(* IEC 61131-3 sources: Yaha/Documentation/Infomaterial/OSCAT/pcworx_basic_333/module_export (part 5) *)

(* ---- MATRIX.ST ---- *)
(*@PROPERTIES_EX@
TYPE: POU
LOCALE: 0
IEC_LANGUAGE: ST
PLC_TYPE: independent
PROC_TYPE: independent
GROUP: LOGIC.OTHER
*)
(*@KEY@:DESCRIPTION*)
version 1.3	26 oct. 2008
programmer 	hugo
tested by	oscat

MATRIX is a matrix keyboard encoder for 4 rows and up to 5 columns.
matrix can send a code while a key is pressed and it sends another code while a key is released when the setup variable 'release' is set to true.
the setup variable release is false the code is only sent when the key is pressed.
the output byte holds the 5 columns in the lowest bits 0..2  and the row number in bits 4..6, while bit 7 is true for a key pressed and false for a key released.
(*@KEY@:END_DESCRIPTION*)
FUNCTION_BLOCK MATRIX

(*Group:Default*)

VAR_INPUT
	X1 :	BOOL;
	X2 :	BOOL;
	X3 :	BOOL;
	X4 :	BOOL;
	X5 :	BOOL;
	RELEASE :	BOOL;
END_VAR

VAR_OUTPUT
	CODE :	BYTE;
	TP :	BOOL;
	Y1 :	BOOL := TRUE;
	Y2 :	BOOL;
	Y3 :	BOOL;
	Y4 :	BOOL;
END_VAR

VAR
	line :	BYTE;
	X :	oscat_arb_0_3;(*scan line inputs*)
	L :	oscat_arb_0_3;(*scan line status*)
	i :	INT;
	temp :	BYTE;
	temp2 :	BYTE;
	L_temp :	BYTE;
	temp_bit :	BOOL;
	in_temp :	INT;
END_VAR

(*@KEY@: WORKSHEET
NAME: MATRIX
IEC_LANGUAGE: ST
*)
TP := FALSE;
code := BYTE#0;

(* read scan lines *)
in_temp := _BYTE_TO_INT(line);
temp := X[in_temp];  (* X[LINE] umkopieren *)

temp:=BIT_LOAD_B(temp,X1,0); (* X[line].0 := X1; *)
temp:=BIT_LOAD_B(temp,X2,1); (* X[line].1 := X2; *)
temp:=BIT_LOAD_B(temp,X3,2); (* X[line].2 := X3; *)
temp:=BIT_LOAD_B(temp,X4,3); (* X[line].3 := X4; *)
temp:=BIT_LOAD_B(temp,X5,4); (* X[line].4 := X5; *)

X[in_temp] := temp; (* X[LINE] zurückkopieren *)

(* compare for change *)
FOR i := 0 TO 3 DO
	IF X[i] <> L[i] THEN
		(* scan line information has changed code need to be found and generated *)
		temp   := x[i] XOR L[i];
        temp2  := X[i];
        L_temp := L[i];

        IF BIT_OF_DWORD(BYTE_TO_DWORD(temp),0) THEN (* temp.X0 *)
			code := BYTE#1;
            temp_bit := BIT_OF_DWORD(BYTE_TO_DWORD(temp2),0);   (* X[i].X0 *)
            code := BIT_LOAD_B(code,temp_bit,7);     			(* code.X7 *)
            L_temp := BIT_LOAD_B(L_temp,temp_bit,0); 			(* L[i].X0 *)
		ELSIF BIT_OF_DWORD(BYTE_TO_DWORD(temp),1) THEN          (* temp.X1 *)
			code := BYTE#2;
            temp_bit := BIT_OF_DWORD(BYTE_TO_DWORD(temp2),1);   (* X[i].X1 *)
            code := BIT_LOAD_B(code,temp_bit,7);     			(* code.X7 *)
            L_temp := BIT_LOAD_B(L_temp,temp_bit,1); 			(* L[i].X1 *)
		ELSIF BIT_OF_DWORD(BYTE_TO_DWORD(temp),2) THEN          (* temp.X2 *)
			code := BYTE#3;
            temp_bit := BIT_OF_DWORD(BYTE_TO_DWORD(temp2),2);   (* X[i].X2 *)
            code := BIT_LOAD_B(code,temp_bit,7);     			(* code.X7 *)
            L_temp := BIT_LOAD_B(L_temp,temp_bit,2); 			(* L[i].X2 *)
		ELSIF BIT_OF_DWORD(BYTE_TO_DWORD(temp),3) THEN          (* temp.X3 *)
			code := BYTE#4;
            temp_bit := BIT_OF_DWORD(BYTE_TO_DWORD(temp2),3);   (* X[i].X3 *)
            code := BIT_LOAD_B(code,temp_bit,7);     			(* code.X7 *)
            L_temp := BIT_LOAD_B(L_temp,temp_bit,3); 			(* L[i].X3 *)
		ELSIF BIT_OF_DWORD(BYTE_TO_DWORD(temp),4) THEN          (* temp.X4 *)
			code := BYTE#5;
            temp_bit := BIT_OF_DWORD(BYTE_TO_DWORD(temp2),4);   (* X[i].X4 *)
            code := BIT_LOAD_B(code,temp_bit,7);     			(* code.X7 *)
            L_temp := BIT_LOAD_B(L_temp,temp_bit,4); 			(* L[i].X4 *)
		END_IF;
        L[i] := L_temp;
		TP := TRUE;
        code := (code AND BYTE#2#1000_1111) OR SHL(LINE AND BYTE#2#0000_0111,4);
        (* obere zeile enspricht: Code.X4 := Line.X0; /  Code.X5 := Line.X1; / Code.X6 := Line.X2; *)

		(* check if release codes need to be killed *)
		IF NOT release AND code < BYTE#127 THEN
			code := BYTE#0;
			TP := FALSE;
		END_IF;
        EXIT;
	END_IF;
END_FOR;

(* increment scan line every cycle *)
line := INT_TO_BYTE(_BYTE_TO_INT(line) + 1) AND BYTE#2#0000_0011;
temp := SHL(BYTE#1,_BYTE_TO_INT(line));

Y1 := BIT_OF_DWORD(BYTE_TO_DWORD(temp),0); (* temp.0 *)
Y2 := BIT_OF_DWORD(BYTE_TO_DWORD(temp),1); (* temp.1 *)
Y3 := BIT_OF_DWORD(BYTE_TO_DWORD(temp),2); (* temp.2 *)
Y4 := BIT_OF_DWORD(BYTE_TO_DWORD(temp),3); (* temp.3 *)

(* revision history
hm		10.6.2007	rev 1.0
	original version

hm		11.9.2007	rev 1.1
	deleted unused variables k and old_code

hm		23.12.2007	rev 1.2
	added exit statement in for loop instead of i:=5

hm		26. oct. 2008	rev 1.3
	code optimized

*)
(*@KEY@: END_WORKSHEET *)
END_FUNCTION_BLOCK

(* ---- MESSAGE_4R.ST ---- *)
(*@PROPERTIES_EX@
TYPE: POU
LOCALE: 0
IEC_LANGUAGE: ST
PLC_TYPE: independent
PROC_TYPE: independent
GROUP: STRINGS
*)
(*@KEY@:DESCRIPTION*)
version 1.1	27. oct. 2008
programmer 	hugo
tested by	tobias

this function generates a rotation meassage with up to 4 strings.
on each rising edge of EN the next message in line will be displayed.
when EN stays high longer then one cycle, the next message will be displayed automatically after the time T1 is elapsed.
the output MX is the generated message and CX is a counter 0..3 signaling the current message displayed.
the displayed messages are 0 .. MM.
(*@KEY@:END_DESCRIPTION*)
FUNCTION_BLOCK MESSAGE_4R

(*Group:Default*)

VAR_INPUT
	M0 :	STRING;
	M1 :	STRING;
	M2 :	STRING;
	M3 :	STRING;
	MM :	INT := 3;
	ENQ :	BOOL := TRUE;
	CLK :	BOOL := TRUE;
	T1 :	TIME := T#3s;
END_VAR

VAR_OUTPUT
	MX :	STRING;
	MN :	INT;
	TR :	BOOL;
END_VAR

VAR
	timer :	TON;
	edge :	BOOL;
END_VAR

(*@KEY@: WORKSHEET
NAME: MESSAGE_4R
IEC_LANGUAGE: ST
*)
(* check for rising edge on EN *)
TR := FALSE;
IF ENQ THEN
	IF (NOT edge AND clk) OR timer.q THEN
			MN := INC1(MN, MM);
			TR := TRUE;
			timer(in := FALSE);
			CASE MN OF
				0 : MX := M0;
				1 : MX := M1;
				2 : MX := M2;
				3 : MX := M3;
			END_CASE;
	END_IF;
	edge := clk;
	timer( in := CLK, pt := T1);
ELSE
	MX := '';
	MN := 0;
END_IF;

(* revision history
hm	8. oct. 2008	rev 1.0
	original version

hm	27. oct. 2008	rev 1.1
	changed _INC to INC1

*)
(*@KEY@: END_WORKSHEET *)
END_FUNCTION_BLOCK

(* ---- MESSAGE_8.ST ---- *)
(*@PROPERTIES_EX@
TYPE: POU
LOCALE: 0
IEC_LANGUAGE: ST
PLC_TYPE: independent
PROC_TYPE: independent
GROUP: STRINGS
*)
(*@KEY@:DESCRIPTION*)
version 1.1	29. mar. 2008
programmer 	hugo
tested by	tobias

this function generates one out of 4 messages specified by S1 .. S8.
the selected message will be presented at the output M.
In1 has higher priority then In2 which has higher priority then IN3 and in8 has the lowest priority.
(*@KEY@:END_DESCRIPTION*)
FUNCTION_BLOCK MESSAGE_8

(*Group:Default*)

VAR_INPUT
	IN1 :	BOOL;
	IN2 :	BOOL;
	IN3 :	BOOL;
	IN4 :	BOOL;
	IN5 :	BOOL;
	IN6 :	BOOL;
	IN7 :	BOOL;
	IN8 :	BOOL;
	S1 :	STRING;
	S2 :	STRING;
	S3 :	STRING;
	S4 :	STRING;
	S5 :	STRING;
	S6 :	STRING;
	S7 :	STRING;
	S8 :	STRING;
END_VAR

VAR_OUTPUT
	M :	STRING;
END_VAR

(*@KEY@: WORKSHEET
NAME: MESSAGE_8
IEC_LANGUAGE: ST
*)
(* check if an alarm is present if yes set the output M otherwise clear M *)
IF in1 THEN
	M := S1;
ELSIF in2 THEN
	M := S2;
ELSIF in3 THEN
	M := S3;
ELSIF in4 THEN
	M := S4;
ELSIF in5 THEN
	M := S5;
ELSIF in6 THEN
	M := S6;
ELSIF in7 THEN
	M := S7;
ELSIF in8 THEN
	M := S8;
ELSE
	M := '';
END_IF;

(* revision history
hm	26.12.2007		rev 1.0
	original version

hm	29. mar. 2008	rev 1.1
	changed STRING to STRING(STRING_LENGTH)
*)
(*@KEY@: END_WORKSHEET *)
END_FUNCTION_BLOCK

(* ---- METER.ST ---- *)
(*@PROPERTIES_EX@
TYPE: POU
LOCALE: 0
IEC_LANGUAGE: ST
PLC_TYPE: independent
PROC_TYPE: independent
GROUP: ENGINEERING.MEASUREMENTS
*)
(*@KEY@:DESCRIPTION*)
version 1.4	8. mar. 2009
programmer 	oscat
tested BY	oscat

METER measures usage of power or similar values the output MX is the sum of the inputs over time.
MX := sum over time of (I1 * P1 + I2 * P2)/D.
a simple example is the consumption counter for a 2 stage oil burner where stage 1 is 10KW and stage 2 is 20KW.
I1 and I2 decide which value is accounted for, I1 = True only counts P1, I2 is True counts P2
and I1 and I2 is true counts P1 and P2.
the meter can be used for all kind of consumption meters. P1 and P2 can change on the fly.

(*@KEY@:END_DESCRIPTION*)
FUNCTION_BLOCK METER

(*Group:Default*)

VAR_INPUT
	M1 :	REAL;
	M2 :	REAL;
	I1 :	BOOL;
	I2 :	BOOL;
	D :	REAL := 1.0;
	RST :	BOOL;
END_VAR

VAR_IN_OUT
	MX :	REAL;
END_VAR

VAR RETAIN
	MR :	REAL2;
END_VAR

VAR
	MX1 :	REAL;(*current consumption value on M1 and M2*)
	MX2 :	REAL;(*current consumption value on M1 and M2*)
	tx :	UDINT;
	last :	UDINT;
	tc :	REAL;
	init :	BOOL;
	T_PLC_MS :	T_PLC_MS;
	R2_ADD :	R2_ADD;
END_VAR

(*@KEY@: WORKSHEET
NAME: METER
IEC_LANGUAGE: ST
*)
(* measure the last cycle time and make sure we onle execute once every millisecond *)
T_PLC_MS();
tx:= T_PLC_MS.T_PLC_MS;
IF NOT init THEN
	init := TRUE;
	last := tx;
	mr.RX := mx;
	mr.R1 := 0.0;
ELSIF tx = last THEN
	RETURN;
ELSE
	tc := UDINT_TO_REAL(tx - last) * 0.001;
END_IF;
last := tx;

(* reset *)
IF rst THEN
	mr.R1 := 0.0;
	mr.RX := 0.0;
ELSE
	(* current consumption measurement *)
	MX1 := SEL(I1,0.0,M1);
	MX2 := SEL(I2,0.0,M2);
	(* add up the current values in a double real *)
	R2_ADD(X:=MR,Y:=(SEL(I1,0.0,mx1) + SEL(I2, 0.0, mx2)) / D * TC);
	MR:=R2_ADD.R2_ADD;
	(* set the current output value *)
	MX := mr.RX;
END_IF;

(* revision history

hm	16. sep.2007		rev 1.0
	original version

hm	7. feb 2008		rev 1.1
	use new version of ft_int to avoid a counting stop at high values
	deleted unnecessary limits

hm	24. mar. 2008		rev 1.2
	use data_type real2 to extend accuracy to 15 digits total
	do not use ft_int which adds unnecessary overhead

hm	8. feb. 2009		rev 1.3
	changed mx to be I/O
	make sure calculation works for cycle times < 1 ms

hm	8. mar. 2009	rev 1.4
	last was not updated
	code improvements

*)

(*@KEY@: END_WORKSHEET *)
END_FUNCTION_BLOCK

(* ---- METER_STAT.ST ---- *)
(*@PROPERTIES_EX@
TYPE: POU
LOCALE: 0
IEC_LANGUAGE: ST
PLC_TYPE: independent
PROC_TYPE: independent
GROUP: ENGINEERING.MEASUREMENTS
*)
(*@KEY@:DESCRIPTION*)
version 1.3	18. jul. 2009
programmer 	oscat
tested BY	oscat

METER_STAT runs statistics of a metered value, it calculates the current week, day, month and year consumption and stores the corresponding last day, week, month and year value.

(*@KEY@:END_DESCRIPTION*)
FUNCTION_BLOCK METER_STAT

(*Group:Default*)

VAR_INPUT
	IN :	REAL;
	DI :	UDINT;
	RST :	BOOL;
END_VAR

VAR_IN_OUT
	LAST_DAY :	REAL;
	CURRENT_DAY :	REAL;
	LAST_WEEK :	REAL;
	CURRENT_WEEK :	REAL;
	LAST_MONTH :	REAL;
	CURRENT_MONTH :	REAL;
	LAST_YEAR :	REAL;
	CURRENT_YEAR :	REAL;
END_VAR

VAR RETAIN
	year_start :	REAL;
	month_start :	REAL;
	week_start :	REAL;
	day_start :	REAL;
	last_run :	UDINT;
END_VAR

(*@KEY@: WORKSHEET
NAME: METER_STAT
IEC_LANGUAGE: ST
*)
IF rst THEN
	Last_Day := 0.0;
	Current_Day := 0.0;
	Day_start := IN;
	Last_week := 0.0;
	Current_week := 0.0;
	Week_start := in;
	Last_month := 0.0;
	Current_month := 0.0;
	month_start := in;
	last_year := 0.0;
	current_year := 0.0;
	year_start := in;
ELSE
	Current_Day := IN - Day_Start;
	Current_Week := In - Week_Start;
	Current_Month := IN - Month_Start;
	Current_Year := IN - Year_Start;
END_IF;

IF YEAR_OF_DATE(DI) > YEAR_OF_DATE(last_run) THEN
	(* a new year has started *)
	last_year := current_year;
	current_year := 0.0;
	year_start := in;
	last_month := current_month;
	current_month := 0.0;
	month_start := in;
	last_day := current_day;
	current_day := 0.0;
	day_start := in;
ELSIF MONTH_OF_DATE(DI) > MONTH_OF_DATE(last_run) THEN
	(* a new month has started, january is alrerady done by year change *)
	last_month := current_month;
	current_month := 0.0;
	month_start := in;
	last_day := current_day;
	current_day := 0.0;
	day_start := in;
ELSIF DAY_OF_YEAR(di) > DAY_OF_YEAR(last_run) THEN
	(* day has chaged, first day of year and first day of month has already been taken care of *)
	last_day := current_day;
	current_day := 0.0;
	day_start := in;
END_IF;
IF DAY_OF_WEEK(DI) < DAY_OF_WEEK(last_run) THEN
	(* a new week has started *)
	last_week := current_week;
	current_week := 0.0;
	week_start := in;
END_IF;
last_run := di;

(* revision history
hm	16. sep. 2007	rev 1.0
	original version

hm	7. oct. 2008	rev 1.1
	changed function year_to_year_of_date
	changed function month to month_of_date
	changed function weekday to day_of_week

hm	11. mar. 2009	rev 1.2
	changed real constants to use dot syntax

hm	18. jul. 2009	rev 1.3
	changes all outputs to be I/O
*)

(*@KEY@: END_WORKSHEET *)
END_FUNCTION_BLOCK

(* ---- MIRROR.ST ---- *)
(*@PROPERTIES_EX@
TYPE: POU
LOCALE: 0
IEC_LANGUAGE: ST
PLC_TYPE: independent
PROC_TYPE: independent
GROUP: STRINGS
*)
(*@KEY@:DESCRIPTION*)
version 1.1	29. mar. 2008
programmer 	hugo
tested by	tobias

this function reverses an input string.
(*@KEY@:END_DESCRIPTION*)
FUNCTION_BLOCK MIRROR

(*Group:Default*)

VAR_INPUT
	STR :	STRING;
END_VAR

VAR_OUTPUT
	MIRROR :	STRING;
END_VAR

VAR
	i :	INT;
	st_temp :	STRING;
END_VAR

(*@KEY@: WORKSHEET
NAME: MIRROR
IEC_LANGUAGE: ST
*)
mirror := '';
i := LEN(str);
WHILE i > 0 DO
   st_temp := MID(str,1,i);
   mirror := CONCAT(mirror,st_temp);
   i := i -1;
END_WHILE;

(* revision histroy
hm	4. feb. 2008	rev 1.0
	original release

hm	29. mar. 2008	rev 1.1
	changed STRING to STRING(STRING_LENGTH)
*)
(*@KEY@: END_WORKSHEET *)
END_FUNCTION_BLOCK

(* ---- MONTH_TO_STRING.ST ---- *)
(*@PROPERTIES_EX@
TYPE: POU
LOCALE: 0
IEC_LANGUAGE: ST
PLC_TYPE: independent
PROC_TYPE: independent
GROUP: STRINGS
*)
(*@KEY@:DESCRIPTION*)
version 1.1	19. oct. 2008
programmer 	hugo
tested by	oscat

MONTH_TO_STRING converts an Integer 1..12 into a String with the Names of the corresponding Month.
the decoding is according to the language setup in global vars
(*@KEY@:END_DESCRIPTION*)
FUNCTION_BLOCK MONTH_TO_STRING

(*Group:Default*)

VAR_INPUT
	MTH :	INT;
	LANG :	INT;
	LX :	INT;
END_VAR

VAR_OUTPUT
	MONTH_TO_STRING :	oscat_STRING10;
END_VAR

VAR
	LY :	INT;
	SETUP_MONTHS :	SETUP_MONTHS;
	MONTHS :	oscat_MONTHS;
	SETUP_MONTHS3 :	SETUP_MONTHS3;
	MONTHS3 :	oscat_MONTHS3;
	SETUP_LANGUAGE :	SETUP_LANGUAGE;
	LANGUAGE :	oscat_LANGUAGE;
END_VAR

(*@KEY@: WORKSHEET
NAME: MONTH_TO_STRING
IEC_LANGUAGE: ST
*)
SETUP_MONTHS(MONTHS:=MONTHS);
MONTHS:=SETUP_MONTHS.MONTHS;
SETUP_MONTHS3(MONTHS3:=MONTHS3);
MONTHS3:=SETUP_MONTHS3.MONTHS3;
SETUP_LANGUAGE(LANGUAGE:=LANGUAGE);
LANGUAGE:=SETUP_LANGUAGE.LANGUAGE;

IF LANG = 0 THEN Ly := LANGUAGE.DEFAULT; ELSE ly := MIN(LANG, language.LMAX); END_IF;
IF MTH < 1 OR MTH > 12 THEN
	RETURN;
ELSIF LX = 0 THEN
	MONTH_TO_STRING := MONTHS[ly][MTH];
ELSIF Lx = 3 THEN
	MONTH_TO_STRING := MONTHS3[ly][MTH];
END_IF;

(* revisison history

hm	21. sep. 2008	rev 1.0
	original version

hm	19. oct. 2008	rev 1.1
	changed language setup constants
*)
(*@KEY@: END_WORKSHEET *)
END_FUNCTION_BLOCK

(* ---- OCT_TO_BYTE.ST ---- *)
(*@PROPERTIES_EX@
TYPE: POU
LOCALE: 0
IEC_LANGUAGE: ST
PLC_TYPE: independent
PROC_TYPE: independent
GROUP: STRINGS
*)
(*@KEY@:DESCRIPTION*)
version 1.1	20. sep. 2008
programmer 	hugo
tested by	oscat

OCT_TO_BYTE converts a octagonal string into a byte.
(*@KEY@:END_DESCRIPTION*)
FUNCTION_BLOCK OCT_TO_BYTE

(*Group:Default*)

VAR_INPUT
	OCT :	oscat_STRING10;
END_VAR

VAR_OUTPUT
	OCT_TO_BYTE :	BYTE;
END_VAR

VAR
	i :	INT;
	stop :	INT;
	X :	INT;
END_VAR

(*@KEY@: WORKSHEET
NAME: OCT_TO_BYTE
IEC_LANGUAGE: ST
*)
OCT_TO_BYTE := BYTE#0;
stop := LEN(oct);
FOR I := 1 TO stop DO
	(* read the first character and subtract 48 to get value in decimal 0 = 48 *)
    X := GET_CHAR(oct,I);
	(* calculate the value of the digit *)
	IF X > 47 AND x < 56 THEN
	    OCT_TO_BYTE := SHL_BYTE(OCT_TO_BYTE,3) OR INT_TO_BYTE(X - 48);
	END_IF;
END_FOR;

(* revision histroy
hm	18. jun. 2008	rev 1.0
	original release

hm	20. sep. 2008	rev 1.1
	changed length of input string from 20 to 10

*)
(*@KEY@: END_WORKSHEET *)
END_FUNCTION_BLOCK

(* ---- OCT_TO_DWORD.ST ---- *)
(*@PROPERTIES_EX@
TYPE: POU
LOCALE: 0
IEC_LANGUAGE: ST
PLC_TYPE: independent
PROC_TYPE: independent
GROUP: STRINGS
*)
(*@KEY@:DESCRIPTION*)
version 1.0	18. jun 2008
programmer 	hugo
tested by	oscat

OCT_TO_DWORD converts a octagonal string into a dword.
(*@KEY@:END_DESCRIPTION*)
FUNCTION_BLOCK OCT_TO_DWORD

(*Group:Default*)

VAR_INPUT
	OCT :	oscat_STRING20;
END_VAR

VAR_OUTPUT
	OCT_TO_DWORD :	DWORD;
END_VAR

VAR
	i :	INT;
	stop :	INT;
	X :	INT;
END_VAR

(*@KEY@: WORKSHEET
NAME: OCT_TO_DWORD
IEC_LANGUAGE: ST
*)
OCT_TO_DWORD := DWORD#0;
stop := LEN(oct);
FOR I := 1 TO stop DO
	(* read the first character and subtract 48 to get value in decimal 0 = 48 *)
    X := GET_CHAR(oct,I);
	(* calculate the value of the digit *)
	IF X > 47 AND x < 56 THEN
	    OCT_TO_DWORD := SHL_DWORD(OCT_TO_DWORD,3) OR INT_TO_DWORD(X - 48);
	END_IF;
END_FOR;

(* revision histroy
hm	2.10.2007		rev 1.0
	original release

hm	19.11.2007		rev 1.1
	changed type of function from int to dword

hm 	4. mar 2008		rev 1.2
	added support for a..f and return 0 for invalid string

hm	29. mar. 2008	rev 1.3
	changed STRING to STRING(8)

hm	18. jun. 2008	rev 1.4
	changed input hex to STRING(20)
	function now ignores wrong characters
*)
(*@KEY@: END_WORKSHEET *)
END_FUNCTION_BLOCK

(* ---- ONTIME.ST ---- *)
(*@PROPERTIES_EX@
TYPE: POU
LOCALE: 0
IEC_LANGUAGE: ST
PLC_TYPE: independent
PROC_TYPE: independent
GROUP: ENGINEERING.MEASUREMENTS
*)
(*@KEY@:DESCRIPTION*)
version 2.5	18. mar. 2011
programmer 	oscat
tested by	tobias

ONTIME measures the ontime of a signal in seconds.
the output SECONDS is of type DWORD which results in a total measurement range of 1 second up to 136 years.
internally ontime works with a resolution of milliseconds
(*@KEY@:END_DESCRIPTION*)
FUNCTION_BLOCK ONTIME

(*Group:Default*)

VAR_INPUT
	IN :	BOOL;
	RST :	BOOL;
END_VAR

VAR_IN_OUT
	SECONDS :	UDINT;
	CYCLES :	UDINT;
END_VAR

VAR
	tx :	UDINT;
	last :	UDINT;
	edge :	BOOL;
	init :	BOOL;
	ms :	UDINT;
	T_PLC_MS :	T_PLC_MS;
END_VAR

(*@KEY@: WORKSHEET
NAME: ONTIME
IEC_LANGUAGE: ST
*)
(* read system time *)
T_PLC_MS();
tx:= T_PLC_MS.T_PLC_MS;

(* make sure the first cycle works correctly *)
IF NOT init THEN
	init := TRUE;
	last := tx;
	ms := UDINT#0;
END_IF;
IF RST THEN
	SECONDS := UDINT#0;
	CYCLES := UDINT#0;
	last := tx;
	ms := UDINT#0;
ELSIF IN THEN
	(* add the current milliseconds *)
	ms := (tx - last) + ms;
	IF ms >= UDINT#1000 THEN
		seconds := seconds + UDINT#1;
		ms := ms - UDINT#1000;
	END_IF;
	cycles := cycles + BOOL_TO_UDINT(NOT edge);
END_IF;
last := tx;
edge := in;

(* revision history
hm 22.2.2007		rev 1.1
	changed VAR RETAIN PERSISTENT to VAR RETAIN for better compatibility
	wago lon contollers do not support persisitent

hm 2.8.2007		rev 1.2
	adding time up in a real number will automatically lead to the point where
	small time scales like the cycle time will be below the resolution of real and therefore
	ontime would not increase in small steps as necessary
	the time is now measured internally in two  dwords and be converted to real only for
	output purposes.
	deleted the variable power because it was unnecessary

hm	16.9.2007		rev 1.3
	changes time() to T_plc_ms() for compatibility reasons

hm	2. dec. 2007	rev 1.4
	chaged code for better performance

hm	16. mar. 2008	rev 1.5
	added type conversions to avoid warnings under codesys 3.0

hm	21. oct. 2008	rev 2.0
	changed module for much better performance and allow for external result storage

hm	10. nov. 2008	rev 2.1
	increased internal resolution to milliseconds

hm	16. nov. 2008	rev 2.2
	changed typecast to avoid warnings

hm	17. dec. 2008	rev 2.3
	fixed an error when in would be true for more then 49 days

hm	17. jan 2011	rev 2.4
	init will not clear seconds and cycles, only rst clears these values

hm	18. mar. 2011	rev 2.5
	reset was not working

*)

(*@KEY@: END_WORKSHEET *)
END_FUNCTION_BLOCK

(* ---- PARSET.ST ---- *)
(*@PROPERTIES_EX@
TYPE: POU
LOCALE: 0
IEC_LANGUAGE: ST
PLC_TYPE: independent
PROC_TYPE: independent
GROUP: ENGINEERING.AUTOMATION
*)
(*@KEY@:DESCRIPTION*)
version 1.1	16. mar. 2008
programmer 	hugo
tested by		tobias

parset selects on of 4 parameter sets adressed by the inputs A0 and A1. if TC is specified, the change of the outputs
is ramped by the time tc
(*@KEY@:END_DESCRIPTION*)
FUNCTION_BLOCK PARSET

(*Group:Default*)

VAR_INPUT
	A0 :	BOOL;
	A1 :	BOOL;
	X01 :	REAL;
	X02 :	REAL;
	X03 :	REAL;
	X04 :	REAL;
	X11 :	REAL;
	X12 :	REAL;
	X13 :	REAL;
	X14 :	REAL;
	X21 :	REAL;
	X22 :	REAL;
	X23 :	REAL;
	X24 :	REAL;
	X31 :	REAL;
	X32 :	REAL;
	X33 :	REAL;
	X34 :	REAL;
	TC :	TIME;
END_VAR

VAR_OUTPUT
	P1 :	REAL;
	P2 :	REAL;
	P3 :	REAL;
	P4 :	REAL;
END_VAR

VAR
	X :	oscat_parset;
	S1 :	REAL;
	S2 :	REAL;
	S3 :	REAL;
	S4 :	REAL;
	tx :	UDINT;
	last :	UDINT;
	start :	BOOL;
	set :	BYTE;
	set2 :	INT;
	init :	BOOL;
	T_PLC_MS :	T_PLC_MS;
END_VAR

(*@KEY@: WORKSHEET
NAME: PARSET
IEC_LANGUAGE: ST
*)
(* read system_time *)
T_PLC_MS();
tx:= T_PLC_MS.T_PLC_MS;

(* init sequence *)
IF NOT init THEN
    set:=BIT_LOAD_B(set,NOT A0,0); (* set.X0 := NOT A0; *)
	init := TRUE;
	X[0][1] := X01;
	X[0][2] := X02;
	X[0][3] := X03;
	X[0][4] := X04;
	X[1][1] := X11;
	X[1][2] := X12;
	X[1][3] := X13;
	X[1][4] := X14;
	X[2][1] := X21;
	X[2][2] := X22;
	X[2][3] := X23;
	X[2][4] := X24;
	X[3][1] := X31;
	X[3][2] := X32;
	X[3][3] := X33;
	X[3][4] := X34;
	P1 := X01;
	P2 := X02;
	P3 := X03;
	P4 := X04;
END_IF;

(* check for input change *)
IF (A0 XOR BIT_OF_DWORD(BYTE_TO_DWORD(set),0)) OR (A1 XOR BIT_OF_DWORD(BYTE_TO_DWORD(set),1)) THEN  (* set.X0  ,  set.X1 *)
	(* a new set is selected *)
    set := BIT_LOAD_B(set,A0,0); (* set.X0 := A0; *)
    set := BIT_LOAD_B(set,A1,1); (* set.X1 := A1; *)

	IF tc > t#0s THEN
		start := TRUE;
		last := tx;
		(* save the step speed for the output changes in S *)
		set2 := _BYTE_TO_INT(set);
		S1 := (X[set2][1] - P1)/TIME_TO_REAL(tc);
		S2 := (X[set2][2] - P2)/TIME_TO_REAL(tc);
		S3 := (X[set2][3] - P3)/TIME_TO_REAL(tc);
		S4 := (X[set2][4] - P4)/TIME_TO_REAL(tc);
	END_IF;
ELSIF start AND tx - last < TIME_TO_UDINT(tc) THEN
	(* ramp the outputs to the new value *)
	set2 := _BYTE_TO_INT(set);
	P1 := X[set2][1] - S1*(TIME_TO_REAL(Tc) - UDINT_TO_REAL(tx + last));
	P2 := X[set2][2] - S2*(TIME_TO_REAL(Tc) - UDINT_TO_REAL(tx + last));
	P3 := X[set2][3] - S3*(TIME_TO_REAL(Tc) - UDINT_TO_REAL(tx + last));
	P4 := X[set2][4] - S4*(TIME_TO_REAL(Tc) - UDINT_TO_REAL(tx + last));
ELSE
	(* make sure outputs match the correct set values *)
	set2 := _BYTE_TO_INT(set);
	start := FALSE;
	P1 := X[set2][1];
	P2 := X[set2][2];
	P3 := X[set2][3];
	P4 := X[set2][4];
END_IF;

(* revision history
hm	2.11.2007		rev 1.0
	original version

hm	16. mar. 2008	rev 1.1
	added type conversions to avoid warnings under codesys 3.0

*)
(*@KEY@: END_WORKSHEET *)
END_FUNCTION_BLOCK

(* ---- PARSET2.ST ---- *)
(*@PROPERTIES_EX@
TYPE: POU
LOCALE: 0
IEC_LANGUAGE: ST
PLC_TYPE: independent
PROC_TYPE: independent
GROUP: ENGINEERING.AUTOMATION
*)
(*@KEY@:DESCRIPTION*)
version 1.0	3 nov 2007
programmer 	hugo
tested by	tobias

parset2 selects on of 4 parameter sets depending on the value of X. if TC is specified, the change of the outputs
is ramped by the time TC
(*@KEY@:END_DESCRIPTION*)
FUNCTION_BLOCK PARSET2

(*Group:Default*)

VAR_INPUT
	X :	REAL;
	X01 :	REAL;
	X02 :	REAL;
	X03 :	REAL;
	X04 :	REAL;
	X11 :	REAL;
	X12 :	REAL;
	X13 :	REAL;
	X14 :	REAL;
	X21 :	REAL;
	X22 :	REAL;
	X23 :	REAL;
	X24 :	REAL;
	X31 :	REAL;
	X32 :	REAL;
	X33 :	REAL;
	X34 :	REAL;
	L1 :	REAL;
	L2 :	REAL;
	L3 :	REAL;
	TC :	TIME;
END_VAR

VAR_OUTPUT
	P1 :	REAL;
	P2 :	REAL;
	P3 :	REAL;
	P4 :	REAL;
END_VAR

VAR
	Pset :	parset;
	init :	BOOL;
END_VAR

(*@KEY@: WORKSHEET
NAME: PARSET2
IEC_LANGUAGE: ST
*)
(* init sequence *)
IF NOT init THEN
	init := TRUE;
	pset(TC:=TC, X01:=X01, X02:=X02, X03:=X03, X04:=X04, X11:=X11, X12:=X12, X13:=X13, X14:=X14, X21:=X21, X22:=X22, X23:=X23, X24:=X24, X31:=X31, X32:=X32, X33:=X33, X34:=X34);
END_IF;
IF ABS(X) < L1 THEN
	pset(A0 := FALSE, A1 := FALSE);
ELSIF ABS(X) < L2 THEN
	pset(A0 := TRUE, A1 := FALSE);
ELSIF ABS(x) < L3 THEN
	pset(A0 := FALSE, A1 := TRUE);
ELSE
	pset(A0 := TRUE, A1 := TRUE);
END_IF;
P1 := pset.P1;
P2 := pset.P2;
P3 := pset.P3;
P4 := pset.P4;

(* revision history
hm		3.11.2007		rev 1.0
*)
(*@KEY@: END_WORKSHEET *)
END_FUNCTION_BLOCK

(* ---- PERIOD2.ST ---- *)
(*@PROPERTIES_EX@
TYPE: POU
LOCALE: 0
IEC_LANGUAGE: ST
PLC_TYPE: independent
PROC_TYPE: independent
GROUP: TIME_DATE
*)
(*@KEY@:DESCRIPTION*)
version 1.0	27. apr. 2008
programmer 	hugo
tested by	tobias

PERIOD2 checks if DX is within one of 4 periods and sets the output true if so.
(*@KEY@:END_DESCRIPTION*)
FUNCTION_BLOCK PERIOD2

(*Group:Default*)

VAR_INPUT
	DP :	oscat_PERIOD2_X;
	DX :	UDINT;
END_VAR

VAR_OUTPUT
	PERIOD2 :	BOOL;
END_VAR

(*@KEY@: WORKSHEET
NAME: PERIOD2
IEC_LANGUAGE: ST
*)
PERIOD2 := 	(DX >= DP[0][0] AND DX <= DP[0][1]) OR
			(DX >= DP[1][0] AND DX <= DP[1][1]) OR
			(DX >= DP[2][0] AND DX <= DP[2][1]) OR
			(DX >= DP[3][0] AND DX <= DP[3][1]);

(* revision history

hm		27. apr 2008	rev 1.0
	original version

*)
(*@KEY@: END_WORKSHEET *)
END_FUNCTION_BLOCK

(* ---- PIN_CODE.ST ---- *)
(*@PROPERTIES_EX@
TYPE: POU
LOCALE: 0
IEC_LANGUAGE: ST
PLC_TYPE: independent
PROC_TYPE: independent
GROUP: LOGIC.OTHER
*)
(*@KEY@:DESCRIPTION*)
version 1.0	30. oct. 2008
programmer 	hugo
tested by	oscat

MATRIX_CODE scans the input of a key_pad (MATRIX) for a sequence of characters.
(*@KEY@:END_DESCRIPTION*)
FUNCTION_BLOCK PIN_CODE

(*Group:Default*)

VAR_INPUT
	CB :	BYTE;
	E :	BOOL;
	PIN :	oscat_STRING8;
END_VAR

VAR_OUTPUT
	TP :	BOOL;
END_VAR

VAR
	POS :	INT := 1;
END_VAR

(*@KEY@: WORKSHEET
NAME: PIN_CODE
IEC_LANGUAGE: ST
*)
tp := FALSE;
IF e THEN

	IF CB = INT_TO_BYTE(GET_CHAR(PIN,POS)) THEN
		pos := pos + 1;
		IF pos > LEN(PIN) THEN
			(* proper code is detected *)
			TP := TRUE;
			pos := 1;
		END_IF;
	ELSE
		pos := 1;
	END_IF;
END_IF;

(* revision history
hm	30. oct. 2008	rev 1.0
	original version

*)
(*@KEY@: END_WORKSHEET *)
END_FUNCTION_BLOCK

(* ---- POLYNOM_INT.ST ---- *)
(*@PROPERTIES_EX@
TYPE: POU
LOCALE: 0
IEC_LANGUAGE: ST
PLC_TYPE: independent
PROC_TYPE: independent
GROUP: MATHEMATICAL.FUNCTIONS
*)
(*@KEY@:DESCRIPTION*)
version 1.3	10. mar. 2009
programmer 	oscat
tested BY	oscat

POLYNOM_INT calculates an output based on a Polynom interpolation of up to 5 coordinates given in an array
the indut coordinates have to start at the lowest array position and must be sorted ba ascending X values.

(*@KEY@:END_DESCRIPTION*)
FUNCTION_BLOCK POLYNOM_INT

(*Group:Default*)

VAR_INPUT
	X :	REAL;
	XY :	oscat_Polynom_XY;
END_VAR

VAR
	XY2 :	oscat_Polynom_XY;
END_VAR

VAR_INPUT
	PTS :	INT;
END_VAR

VAR_OUTPUT
	POLYNOM_INT :	REAL;
END_VAR

VAR
	I :	INT;
	J :	INT;
	J_1 :	INT;
	J_I :	INT;
	INIT :	BOOL;
END_VAR

(*@KEY@: WORKSHEET
NAME: POLYNOM_INT
IEC_LANGUAGE: ST
*)
(*make sure n is bound within the array size *)
pts := MIN_INT(pts, 5);

(* this part is only to calculate the polynom parameters, which are then stores in the Y array
	the array values, it is not needed during runtime, unless the parameters will change during runtime
	the remaining code without this setup code can be used within a function to calculate specific functions
	the content of the arrays is then used as constant values within the function *)

IF (init = FALSE) THEN
	init := TRUE;

    (* Daten kopieren *)
	FOR i := 1 TO pts DO
       	FOR j := 0 TO 1 DO
           		XY2[i][j] := XY[i][j];
		END_FOR;
	END_FOR;

	FOR i := 1 TO pts DO
        J := pts;
		WHILE (J >= i+1) DO
          j_i := j-i;
		  j_1 := J-1;
          XY2[j][1] := (XY2[j][1] - XY2[j_1][1]) / (XY2[j][0] - XY2[j_i][0]);
          j := j - 1;
		END_WHILE;
	END_FOR;
END_IF;

(* this part is the actual calculation *)
i := pts;
POLYNOM_INT := 0.0;

WHILE (i >= 1) DO
  POLYNOM_INT := POLYNOM_INT * (X - XY2[i][0]) + XY2[i][1];
  i := i - 1;
END_WHILE;

(* revision history
hm	8. okt 2007	rev 1.0
	original version

hm	17. dec 2007	rev 1.1
	init makes no sense for a function

hm	22. feb 2008	rev 1.2
	improved performance

hm	10. mar. 2009	rev 1.3
	changed syntax of real constants to 0.0

*)
(*@KEY@: END_WORKSHEET *)
END_FUNCTION_BLOCK

(* ---- PRESSURE.ST ---- *)
(*@PROPERTIES_EX@
TYPE: POU
LOCALE: 0
IEC_LANGUAGE: ST
PLC_TYPE: independent
PROC_TYPE: independent
GROUP: ENGINEERING.CONVERSION
*)
(*@KEY@:DESCRIPTION*)
version 1.1	11. mar. 2009
programmer 	hugo
tested by	oscat

this function converts different pressure units
any unused input can simply be left open.
different inputs connected at the same time will be added up.
(*@KEY@:END_DESCRIPTION*)
FUNCTION_BLOCK PRESSURE

(*Group:Default*)

VAR_INPUT
	MWS :	REAL;
	TORR :	REAL;
	ATT :	REAL;
	ATM :	REAL;
	PA :	REAL;
	BAR :	REAL;
END_VAR

VAR_OUTPUT
	YMWS :	REAL;
	YTORR :	REAL;
	YATT :	REAL;
	YATM :	REAL;
	YPA :	REAL;
	YBAR :	REAL;
END_VAR

(*@KEY@: WORKSHEET
NAME: PRESSURE
IEC_LANGUAGE: ST
*)
Ybar := bar +
		pa * 1.0E-5 +
		0.980665 * att +
		1.01325 * atm +
		0.001333224 * torr +
		0.0980665 * mws;
Ymws := ybar * 10.1971621297793;
Ytorr := ybar * 750.0615050434140;
Yatt := ybar * 1.0197162129779;
yatm := ybar * 0.9869232667160;
Ypa := ybar * 100000.0;

(*
Druck, Pascal Pa 1 Pa = 1 N/m2 = 1 kg/(s2 �E m) . 0,75 �E 10.2 mmHg
mechanische 1 MPa = 1 N/mm2 . fur Festigkeitsangaben
Spannung Bar bar 1 bar = 105 Pa = 103 mbar = 105 kg/(s2 �E m)
Millimeter- mmHg 1 mmHg = 133,322 Pa = 1,333 22 mbar
Quecksilbersaule . nur in Heilkunde zulassig
physik. Atmosphare atm 1 atm = 1,013 25 bar
techn. Atmosphare at 1 at = 1 kp/cm2 = 0,980665 bar
Torr Torr 1 Torr = (101325/760) Pa = 1,333224 mbar
Meter-Wassersaule mWS 1 mWS = 9806,65 Pa = 98,0665 mbar
psi lbf/in2 1 lbf/in2 = 68,947 57 mbar = 6894,757 Pa

*)

(* revision history

hm	27. mar. 2007	rev 1.0
	original version

hm	11. mar. 2009	rev 1.1
	improved code

*)
(*@KEY@: END_WORKSHEET *)
END_FUNCTION_BLOCK

(* ---- PWM_DC.ST ---- *)
(*@PROPERTIES_EX@
TYPE: POU
LOCALE: 0
IEC_LANGUAGE: ST
PLC_TYPE: independent
PROC_TYPE: independent
GROUP: ENGINEERING.SIGNAL_GENERATORS
*)
(*@KEY@:DESCRIPTION*)
version 1.4	11. mar. 2009
programmer 	oscat
tested BY	oscat

this signal generator generates a square wave signal which is specified by the frequency and the duty cycle

(*@KEY@:END_DESCRIPTION*)
FUNCTION_BLOCK PWM_DC

(*Group:Default*)

VAR_INPUT
	F :	REAL;
	DC :	REAL;
END_VAR

VAR_OUTPUT
	Q :	BOOL;
END_VAR

VAR
	clk :	CLK_Prg;
	pulse :	TP_X;
	tmp :	REAL;
END_VAR

(*@KEY@: WORKSHEET
NAME: PWM_DC
IEC_LANGUAGE: ST
*)
IF F > 0.0 THEN
	tmp := 1000.0/F;
	CLK(PT := REAL_TO_TIME(tmp));
	Pulse(in := clk.Q, pt := REAL_TO_TIME(tmp*DC));
	Q := pulse.Q;
END_IF;

(* revision history

hm	25. feb 2007	rev 1.1
	recoded in st for better performance and better portability

hm	27. nov 2007	rev 1.2
	avoid divide by 0 when F = 0

hm	19. oct. 2008	rev 1.3
	changed type TP_R to TP_X because of name change
	improved performance

hm	11. mar. 2009	rev 1.4
	changed real constants to use dot syntax

*)
(*@KEY@: END_WORKSHEET *)
END_FUNCTION_BLOCK

(* ---- PWM_PW.ST ---- *)
(*@PROPERTIES_EX@
TYPE: POU
LOCALE: 0
IEC_LANGUAGE: ST
PLC_TYPE: independent
PROC_TYPE: independent
GROUP: ENGINEERING.SIGNAL_GENERATORS
*)
(*@KEY@:DESCRIPTION*)
version 1.5	11. mar. 2009
programmer 	oscat
tested BY	oscat

this signal generator generates a square wave signal which is specified by the frequency and the pulse width.

(*@KEY@:END_DESCRIPTION*)
FUNCTION_BLOCK PWM_PW

(*Group:Default*)

VAR_INPUT
	F :	REAL;
	PW :	TIME;
END_VAR

VAR_OUTPUT
	Q :	BOOL;
END_VAR

VAR
	clk :	CLK_Prg;
	pulse :	TP_X;
END_VAR

(*@KEY@: WORKSHEET
NAME: PWM_PW
IEC_LANGUAGE: ST
*)
IF F > 0.0 THEN
	CLK(PT := REAL_TO_TIME(1000.0 / F));
	Pulse(in := clk.Q, pt := pw);
	Q := pulse.Q;
END_IF;

(* revision history

hm	25. feb 2007	rev 1.1
	recoded in st for better performance and better portability

hm	27. nov 2007	rev 1.2
	avoid divide by 0 when F = 0

hm	9. dec 2007		rev 1.3
	corrected an error with F = 0

hm	19. oct. 2008	rev 1.4
	changed type tp_r to TP_x brecause of name change

hm	11. mar. 2009	rev 1.5
	changed real constants to use dot syntax

*)
(*@KEY@: END_WORKSHEET *)
END_FUNCTION_BLOCK

(* ---- R2_ABS.ST ---- *)
(*@PROPERTIES_EX@
TYPE: POU
LOCALE: 0
IEC_LANGUAGE: ST
PLC_TYPE: independent
PROC_TYPE: independent
GROUP: MATHEMATICAL.DOUBLE_PRECISION
*)
(*@KEY@:DESCRIPTION*)
version 1.1	10. mar. 2009
programmer 	hugo
tested by	tobias

R2_abs returns the absulute value of a double precision real.
(*@KEY@:END_DESCRIPTION*)
FUNCTION_BLOCK R2_ABS

(*Group:Default*)

VAR_INPUT
	X :	REAL2;
END_VAR

VAR_OUTPUT
	R2_ABS :	REAL2;
END_VAR

(*@KEY@: WORKSHEET
NAME: R2_ABS
IEC_LANGUAGE: ST
*)
IF X.RX >= 0.0 THEN
	R2_ABS.RX := X.RX;
	R2_ABS.R1 := X.R1;
ELSE
	R2_ABS.RX := -X.RX;
	R2_ABS.R1 := -X.R1;
END_IF;

(* revision history
hm	21. mar. 2008	rev 1.0
	original version

hm	10. mar. 2009 rev 1.1
	real constants updated to new systax using dot

*)
(*@KEY@: END_WORKSHEET *)
END_FUNCTION_BLOCK

(* ---- R2_ADD.ST ---- *)
(*@PROPERTIES_EX@
TYPE: POU
LOCALE: 0
IEC_LANGUAGE: ST
PLC_TYPE: independent
PROC_TYPE: independent
GROUP: MATHEMATICAL.DOUBLE_PRECISION
*)
(*@KEY@:DESCRIPTION*)
version 1.0	20. mar. 2008
programmer 	hugo
tested by	tobias

R2_add adds a real to a double real which extends the accuracy of a real to twice as many digits
(*@KEY@:END_DESCRIPTION*)
FUNCTION_BLOCK R2_ADD

(*Group:Default*)

VAR_INPUT
	X :	REAL2;
	Y :	REAL;
END_VAR

VAR_OUTPUT
	R2_ADD :	REAL2;
END_VAR

VAR
	temp :	REAL;
END_VAR

(*@KEY@: WORKSHEET
NAME: R2_ADD
IEC_LANGUAGE: ST
*)
temp := X.RX;
R2_ADD.RX := Y + X.R1 + X.RX;
R2_ADD.R1 := temp - R2_ADD.RX + Y + X.R1;

(* revision history
hm		20.3.2008	rev 1.0
	original version

*)
(*@KEY@: END_WORKSHEET *)
END_FUNCTION_BLOCK

(* ---- R2_ADD2.ST ---- *)
(*@PROPERTIES_EX@
TYPE: POU
LOCALE: 0
IEC_LANGUAGE: ST
PLC_TYPE: independent
PROC_TYPE: independent
GROUP: MATHEMATICAL.DOUBLE_PRECISION
*)
(*@KEY@:DESCRIPTION*)
version 1.0	20. mar. 2008
programmer 	hugo
tested by	tobias

R2_add adds a double precision real to a double precision real which extends the accuracy of a real to twice as many digits
(*@KEY@:END_DESCRIPTION*)
FUNCTION_BLOCK R2_ADD2

(*Group:Default*)

VAR_INPUT
	X :	REAL2;
	Y :	REAL2;
END_VAR

VAR_OUTPUT
	R2_ADD2 :	REAL2;
END_VAR

(*@KEY@: WORKSHEET
NAME: R2_ADD2
IEC_LANGUAGE: ST
*)
R2_ADD2.R1 := X.R1 + Y.R1;
R2_ADD2.RX := X.RX + Y.RX;

(* revision history
hm		20.3.2008	rev 1.0
	original version

*)
(*@KEY@: END_WORKSHEET *)
END_FUNCTION_BLOCK

(* ---- R2_DIV.ST ---- *)
(*@PROPERTIES_EX@
TYPE: POU
LOCALE: 0
IEC_LANGUAGE: ST
PLC_TYPE: independent
PROC_TYPE: independent
GROUP: MATHEMATICAL.DOUBLE_PRECISION
*)
(*@KEY@:DESCRIPTION*)
version 1.0	8. mar. 2010
programmer 	hugo
tested by	tobias

R2_div divides a double real by a single real.
(*@KEY@:END_DESCRIPTION*)
FUNCTION_BLOCK R2_DIV

(*Group:Default*)

VAR_INPUT
	X :	REAL2;
	Y :	REAL;
END_VAR

VAR_OUTPUT
	R2_DIV :	REAL2;
END_VAR

(*@KEY@: WORKSHEET
NAME: R2_DIV
IEC_LANGUAGE: ST
*)
R2_DIV.RX := X.RX / Y;
R2_DIV.R1 := X.R1 / Y;

(* revision history
hm	8. mar. 2010	rev 1.0
	original version

*)

(*@KEY@: END_WORKSHEET *)
END_FUNCTION_BLOCK

(* ---- R2_MUL.ST ---- *)
(*@PROPERTIES_EX@
TYPE: POU
LOCALE: 0
IEC_LANGUAGE: ST
PLC_TYPE: independent
PROC_TYPE: independent
GROUP: MATHEMATICAL.DOUBLE_PRECISION
*)
(*@KEY@:DESCRIPTION*)
version 1.0	20. mar. 2008
programmer 	hugo
tested by	tobias

R2_mul multiplies a real with a double real which extends the accuracy of a real to twice as many digits
(*@KEY@:END_DESCRIPTION*)
FUNCTION_BLOCK R2_MUL

(*Group:Default*)

VAR_INPUT
	X :	REAL2;
	Y :	REAL;
END_VAR

VAR_OUTPUT
	R2_MUL :	REAL2;
END_VAR

(*@KEY@: WORKSHEET
NAME: R2_MUL
IEC_LANGUAGE: ST
*)
R2_MUL.RX := X.RX * Y;
R2_MUL.R1 := X.R1 * Y;

(* revision history
hm		20.3.2008	rev 1.0
	original version

*)
(*@KEY@: END_WORKSHEET *)
END_FUNCTION_BLOCK

(* ---- R2_SET.ST ---- *)
(*@PROPERTIES_EX@
TYPE: POU
LOCALE: 0
IEC_LANGUAGE: ST
PLC_TYPE: independent
PROC_TYPE: independent
GROUP: MATHEMATICAL.DOUBLE_PRECISION
*)
(*@KEY@:DESCRIPTION*)
version 1.1	10. mar. 2009
programmer 	hugo
tested by	tobias

R2_set sets a double precision real to a single real value.
(*@KEY@:END_DESCRIPTION*)
FUNCTION_BLOCK R2_SET

(*Group:Default*)

VAR_INPUT
	X :	REAL;
END_VAR

VAR_OUTPUT
	R2_SET :	REAL2;
END_VAR

(*@KEY@: WORKSHEET
NAME: R2_SET
IEC_LANGUAGE: ST
*)
R2_SET.RX := X;
R2_SET.R1 := 0.0;

(* revision history
hm	2. jun. 2008	rev 1.0
	original version

hm	10. mar. 2009	rev 1.1
	real constants updated to new systax using dot

*)
(*@KEY@: END_WORKSHEET *)
END_FUNCTION_BLOCK

(* ---- RDM.ST ---- *)
(*@PROPERTIES_EX@
TYPE: POU
LOCALE: 0
IEC_LANGUAGE: ST
PLC_TYPE: independent
PROC_TYPE: independent
GROUP: MATHEMATICAL.MATHE
*)
(*@KEY@:DESCRIPTION*)
version 1.9	10. mar. 2009
programmer 	hugo
tested by	tobias

this function calculates a pseudo random number
to generate the number it reads the sps timer and calculates a random number between 0 and 1:
in order to use rdm more then once within one sps cycle it need to be called with different seed numbers LAST.

(*@KEY@:END_DESCRIPTION*)
FUNCTION_BLOCK RDM

(*Group:Default*)

VAR_INPUT
	LAST :	REAL;
END_VAR

VAR_OUTPUT
	RDM :	REAL;
END_VAR

VAR
	T_PLC_MS :	T_PLC_MS;
	tn :	DWORD;
	tc :	INT;
END_VAR

(*@KEY@: WORKSHEET
NAME: RDM
IEC_LANGUAGE: ST
*)
T_PLC_MS();
tn := UDINT_TO_DWORD(T_PLC_MS.T_PLC_MS);
tc := Bit_Count(tn);

tn:=BIT_LOAD_DW(tn,BIT_OF_DWORD(tn,2),31); (* tn.31 := tn.2; *)
tn:=BIT_LOAD_DW(tn,BIT_OF_DWORD(tn,5),30); (* tn.30 := tn.5; *)
tn:=BIT_LOAD_DW(tn,BIT_OF_DWORD(tn,4),29); (* tn.29 := tn.4; *)
tn:=BIT_LOAD_DW(tn,BIT_OF_DWORD(tn,1),28); (* tn.28 := tn.1; *)
tn:=BIT_LOAD_DW(tn,BIT_OF_DWORD(tn,0),27); (* tn.27 := tn.0; *)
tn:=BIT_LOAD_DW(tn,BIT_OF_DWORD(tn,7),26); (* tn.26 := tn.7; *)
tn:=BIT_LOAD_DW(tn,BIT_OF_DWORD(tn,6),25); (* tn.25 := tn.6; *)
tn:=BIT_LOAD_DW(tn,BIT_OF_DWORD(tn,3),24); (* tn.24 := tn.3; *)

tn := ROL(tn,Bit_Count(tn)) OR DWORD#16#80000001;
tn := UDINT_TO_DWORD(DWORD_TO_UDINT(tn) MOD UDINT#71474513 + _INT_TO_UDINT(tc) + UDINT#77);
RDM := fract(_DWORD_TO_REAL(tn) / 10000000.0 * (2.71828182845904523536028747135266249 - LIMIT_REAL(0.0,last,1.0)));

(*
pt := ADR(temp);
pt^ := (T_PLC_MS() AND 16#007FFFFF) OR 16#3D000000;
RDM := fract(modR(temp*e+pi1, PI1-last) + modR(temp*PI1+e + last,e-last));
*)

(* revision history
hm		16. jan 2007		rev 1.0
	original version

hm		11. nov 2007		rev 1.1
	changed time() into t_plc_ms()

hm		20. nov 2007		rev 1.2
	changed code of temp calculation to avoid overflow in modr due to resuclt would not fit DINT for high timeer values

hm		5. jan 2008		rev 1.3
	changed calculation of temp to avoid problem with high values of t_plc_ms

hm		2. feb 2008		rev 1.4
	changed algorithm to avoind non iec functions and guarantee more randomness

hm	10. mar. 2008		rev 1.5
	make sure last will be between 0 and 1 to avoid invalid results

hm	16. mar. 2008		rev 1.6
	added conversion for tc to avoid warnings under codesys 3.0

hm	18. may. 2008		rev 1.7
	changed constant E to E1

hm	18. oct. 2008		rev 1.8
	using math constants

hm	10. mar. 2009		rev 1.9
	real constants updated to new systax using dot

*)
(*@KEY@: END_WORKSHEET *)
END_FUNCTION_BLOCK

(* ---- RDM2.ST ---- *)
(*@PROPERTIES_EX@
TYPE: POU
LOCALE: 0
IEC_LANGUAGE: ST
PLC_TYPE: independent
PROC_TYPE: independent
GROUP: MATHEMATICAL.MATHE
*)
(*@KEY@:DESCRIPTION*)
version 1.1	18. oct. 2008
programmer 	hugo
tested by	tobias

this function calculates an integer pseudo random number
the random number will be in the range of low <= rdm2 <= high.
(*@KEY@:END_DESCRIPTION*)
FUNCTION_BLOCK RDM2

(*Group:Default*)

VAR_INPUT
	LAST :	INT;
	LOW :	INT;
	HIGH :	INT;
END_VAR

VAR_OUTPUT
	RDM2 :	INT;
END_VAR

VAR
	rdm :	rdm;
END_VAR

(*@KEY@: WORKSHEET
NAME: RDM2
IEC_LANGUAGE: ST
*)
rdm(last:=fract(INT_TO_REAL(last) * 3.14159265358979323846264338327950288));
RDM2 := TRUNC_INT(rdm.RDM * INT_TO_REAL(high - low + 1)) + low;

(* revision history
hm		29. feb 2008		rev 1.0
	original version

hm		18. oct. 2008		rev 1.1
	using math constants

*)
(*@KEY@: END_WORKSHEET *)
END_FUNCTION_BLOCK

(* ---- RDMDW.ST ---- *)
(*@PROPERTIES_EX@
TYPE: POU
LOCALE: 0
IEC_LANGUAGE: ST
PLC_TYPE: independent
PROC_TYPE: independent
GROUP: MATHEMATICAL.MATHE
*)
(*@KEY@:DESCRIPTION*)
version 1.2	18. oct. 2008
programmer 	hugo
tested by	tobias

this function calculates a DWORD pseudo random number.
(*@KEY@:END_DESCRIPTION*)
FUNCTION_BLOCK RDMDW

(*Group:Default*)

VAR_INPUT
	LAST :	DWORD;
END_VAR

VAR_OUTPUT
	RDMDW :	DWORD;
END_VAR

VAR
	RX :	REAL;
	M :	REAL;
	rdm :	rdm;
END_VAR

(*@KEY@: WORKSHEET
NAME: RDMDW
IEC_LANGUAGE: ST
*)
M := INT_TO_REAL(BIT_COUNT(last));
rdm(last:=FRACT(M*3.14159265358979323846264338327950288));
RX:=rdm.RDM;
RDMDW := SHL_DWORD(_REAL_TO_DWORD(rx*65535.0),16);

rdm(last:=FRACT(M*2.71828182845904523536028747135266249));
RX:=rdm.RDM;
RDMDW := RDMDW OR (_REAL_TO_DWORD(rx*65535.0) AND DWORD#16#0000FFFF);

(* revision history
hm		14. mar 2008		rev 1.0
	original version

hm		18. may. 2008		rev 1.1
	changed constant E to E1

hm		18. oct. 2008		rev 1.2
	using math constants

*)
(*@KEY@: END_WORKSHEET *)
END_FUNCTION_BLOCK

(* ---- REAL_TO_DW.ST ---- *)
(*@PROPERTIES_EX@
TYPE: POU
LOCALE: 0
IEC_LANGUAGE: ST
PLC_TYPE: independent
PROC_TYPE: independent
GROUP: LOGIC.GATE_LOGIC
*)
(*@KEY@:DESCRIPTION*)
version 1.0	18. apr. 2008
programmer 	hugo
tested by	tobias

this function converts a 32 Bit Real to a dword in a bitwise manner.
(*@KEY@:END_DESCRIPTION*)
FUNCTION_BLOCK REAL_TO_DW

(*Group:Default*)

VAR_INPUT
	X :	REAL;
END_VAR

VAR_OUTPUT
	REAL_TO_DW :	DWORD;
END_VAR

VAR
	REAL_TO_BUF :	REAL_TO_BUF;
	i :	INT;
END_VAR

(*@KEY@: WORKSHEET
NAME: REAL_TO_DW
IEC_LANGUAGE: ST
*)
(* REAL_TO_BUF muss mit positiver Flanke gstartet werden darum wird dieser *)
(* einmal mit REQ=0 und dann mit REQ=1 aufgerufen                          *)
(* somit kann in jeden zyklus kopiert werden                               *)

FOR I := 0 TO 1 DO
  REAL_TO_BUF.REQ        := I > 0;
  REAL_TO_BUF.BUF_FORMAT := FALSE;
  REAL_TO_BUF.BUF_OFFS   := DINT#0;
  REAL_TO_BUF.BUF_CNT    := DINT#4;
  REAL_TO_BUF.SRC        := X;
  REAL_TO_BUF.BUFFER     := REAL_TO_DW;
  REAL_TO_BUF();
  X          := REAL_TO_BUF.SRC;
  REAL_TO_DW := REAL_TO_BUF.BUFFER;
END_FOR;
(*@KEY@: END_WORKSHEET *)
END_FUNCTION_BLOCK

(* ---- REAL_TO_FRAC.ST ---- *)
(*@PROPERTIES_EX@
TYPE: POU
LOCALE: 0
IEC_LANGUAGE: ST
PLC_TYPE: independent
PROC_TYPE: independent
GROUP: MATHEMATICAL.MATHE
*)
(*@KEY@:DESCRIPTION*)
version 1.1	06. apr. 2011
programmer 	alexander
tested by	hugo

this function calculates the closest fraction for a real number

(*@KEY@:END_DESCRIPTION*)
FUNCTION_BLOCK REAL_TO_FRAC

(*Group:Default*)

VAR_INPUT
	X :	REAL;
	N :	INT;
END_VAR

VAR_OUTPUT
	REAL_TO_FRAC :	oscat_FRACTION;
END_VAR

VAR
	temp :	DINT;
	sign :	BOOL;
	X_gerundet :	DINT;
	X_ohne_Nachkomma :	REAL;
	Numerator :	DINT := 1;
	Denominator :	DINT := 0;
	Numerator_old :	DINT := 0;
	Denominator_old :	DINT := 1;
END_VAR

(*@KEY@: WORKSHEET
NAME: REAL_TO_FRAC
IEC_LANGUAGE: ST
*)
IF X < 0.0 THEN
	sign := TRUE;								(* Vorzeichen merken *)
	X := ABS(X);								(* Absolutwert berechnen *)
END_IF;

REPEAT
	X_gerundet := REAL_TO_DINT(X);

	(* Zaehler berechnen *)
	temp := numerator * X_gerundet + numerator_old;		(* Zaehler um Vorkammawert erweitern *)
	numerator_old := numerator;							(* Zaehler der letzten Berechnung speichern *)
	numerator := temp;									(* Zaehler dieser Berechnung speichern *)

	(* Nenner berechnen *)
	temp := denominator * X_gerundet + denominator_old;	(* Nenner um Vorkammawert erweitern *)
	denominator_old := denominator;						(* Nenner der letzten Berechnung speichern *)
	denominator := temp;								(* Nenner dieser Berechnung speichern *)

	(* Restwert berechnen *)
	X_ohne_Nachkomma := DINT_TO_REAL(X_gerundet);
	IF X = X_ohne_Nachkomma THEN						(* Bruch geht ohne Rest auf *)
		IF ABS(denominator) <= INT_TO_DINT(N) THEN		(* kein Rundungsfehler *)
			numerator_old := numerator;					(* Numerator_old wird von Funktion zurückgegeben *)
			denominator_old := denominator;				(* Denominator_old wird von Funktion zurückgegeben *)
		END_IF;
		EXIT;											(* keine weitere Berechnung notwendig *)
	ELSE
		X := 1.0 / (X - X_ohne_Nachkomma);				(* Kehrwert vom Rest -> Neuer Bruch *)
	END_IF;

UNTIL
	( ABS(Denominator) > INT_TO_DINT(N))
END_REPEAT;

(* correct sign if X was negative *)
IF sign THEN
	REAL_TO_FRAC.NUMERATOR := -1 * ABS(DINT_TO_INT(numerator_old));
ELSE
	REAL_TO_FRAC.NUMERATOR :=  ABS(DINT_TO_INT(numerator_old));
END_IF;

REAL_TO_FRAC.DENOMINATOR := ABS(DINT_TO_INT(denominator_old));

(* revision history
hm		19. jan. 2011	rev 1.0
	original version

ad		06. apr. 2011	rev 1.1
	optimized code
*)

(*@KEY@: END_WORKSHEET *)
END_FUNCTION_BLOCK

(* ---- REAL_TO_STRF.ST ---- *)
(*@PROPERTIES_EX@
TYPE: POU
LOCALE: 0
IEC_LANGUAGE: ST
PLC_TYPE: independent
PROC_TYPE: independent
GROUP: STRINGS
*)
(*@KEY@:DESCRIPTION*)
version 1.8	2. jan 2012
programmer 	hugo
tested by	oscat

Real_to_strf converts a Real to a fixed length String.
the string will be filles with zeroes to achieve the fixed length N after the decimal separator.
the input parameter specifies the decimal separator to be used in the output string.

(*@KEY@:END_DESCRIPTION*)
FUNCTION_BLOCK REAL_TO_STRF

(*Group:Default*)

VAR_INPUT
	IN :	REAL;
	N :	INT;
	D :	oscat_STRING1;
END_VAR

VAR_OUTPUT
	REAL_TO_STRF :	oscat_STRING20;
END_VAR

VAR
	st_tmp :	oscat_STRING20;
	i :	INT;
END_VAR

(*@KEY@: WORKSHEET
NAME: REAL_TO_STRF
IEC_LANGUAGE: ST
*)
(* LIMIT N to 0 .. 7 *)
N := LIMIT(0,N,7);
(* round the input to N digits and convert to string *)
REAL_TO_STRF := DINT_TO_STRING(_REAL_TO_DINT(ABS(in) * EXP10(INT_TO_REAL(N))),'%d');
(* add zeroes in front to make sure sting is at least 8 digits long *)
FOR i := LEN(REAL_TO_STRF) TO N DO
	st_tmp := REAL_TO_STRF;
	REAL_TO_STRF := CONCAT('0', st_tmp);
END_FOR;
(* add a dot if n > 0 *)
IF n > 0 THEN REAL_TO_STRF := INSERT(REAL_TO_STRF, D, LEN(REAL_TO_STRF) - N); END_IF;
(* add a minus sign if in is negative *)
IF in < 0.0 THEN st_tmp := REAL_TO_STRF; REAL_TO_STRF := CONCAT('-', st_tmp); END_IF;

(* revision history
hm	26 jan 2007	rev 1.0
	original version

hm	20. nov. 2007	rev 1.1
	when N=0 ther will be no dot at the end of the string.

hm	15. dec. 2007	rev 1.2
	changed code for better performance

hm	4. mar. 2008	rev 1.3
	result is now rounded instead of trunc

hm	20. mar. 2008	rev 1.4
	changed trunc to real_to_dint because trunc was generating wrong values on wago 842

hm	29. mar. 2008	rev 1.5
	changed STRING to STRING(20)

hm	4. apr. 2008	rev 1.6
	added variable O to avoid an error uner CoDeSys SP PLCWinNT V2.4

hm	27. feb. 2009	rev 1.7
	added a missing zero for IN < 1

hm 2. jan 2012	rev 1.8
	added input parameter D to specify decimal separator
*)

(*@KEY@: END_WORKSHEET *)
END_FUNCTION_BLOCK

(* ---- REPLACE_ALL.ST ---- *)
(*@PROPERTIES_EX@
TYPE: POU
LOCALE: 0
IEC_LANGUAGE: ST
PLC_TYPE: independent
PROC_TYPE: independent
GROUP: STRINGS
*)
(*@KEY@:DESCRIPTION*)
version 1.1	29. mar. 2008
programmer 	hugo
tested by	tobias

the function findP searches a string str for the occurence of src beginning at the position pos.
(*@KEY@:END_DESCRIPTION*)
FUNCTION_BLOCK REPLACE_ALL

(*Group:Default*)

VAR_INPUT
	STR :	oscat_STRING250;
	SRC :	STRING;
	REP :	STRING;
END_VAR

VAR_OUTPUT
	REPLACE_ALL :	STRING;
END_VAR

VAR
	pos :	INT;
	lp :	INT;
	lx :	INT;
	FINDP :	FINDP;
	st_tmp :	oscat_STRING250;
END_VAR

(*@KEY@: WORKSHEET
NAME: REPLACE_ALL
IEC_LANGUAGE: ST
*)
REPLACE_ALL := str;
lx := LEN(src);
lp := LEN(rep);

FINDP.str := REPLACE_ALL;
FINDP.src := src;
FINDP.pos := 1;
FINDP();
pos := FINDP.FINDP;

WHILE pos > 0 DO
    st_tmp := REPLACE_ALL;
	REPLACE_ALL := REPLACE(st_tmp,rep,lx,pos);

    FINDP.str := REPLACE_ALL;
    FINDP.src := src;
    FINDP.pos := pos + lp;
    FINDP();
    pos := FINDP.FINDP;

END_WHILE;

(* revision histroy
hm	4. feb. 2008	rev 1.0
	original release

hm	29. mar. 2008	rev 1.1
	changed STRING to STRING(STRING_LENGTH)
*)
(*@KEY@: END_WORKSHEET *)
END_FUNCTION_BLOCK

(* ---- REPLACE_CHARS.ST ---- *)
(*@PROPERTIES_EX@
TYPE: POU
LOCALE: 0
IEC_LANGUAGE: ST
PLC_TYPE: independent
PROC_TYPE: independent
GROUP: STRINGS
*)
(*@KEY@:DESCRIPTION*)
version 1.0	14. may. 2008
programmer 	hugo
tested by	hugo

REPLACE_CHARS erstezt alle character die im string src aufgeführt sind mit dem an der selben stelle im string rep gelisteten character.
(*@KEY@:END_DESCRIPTION*)
FUNCTION_BLOCK REPLACE_CHARS

(*Group:Default*)

VAR_INPUT
	STR :	oscat_STRING250;
	SRC :	STRING;
	REP :	STRING;
END_VAR

VAR_OUTPUT
	REPLACE_CHARS :	oscat_STRING250;
END_VAR

VAR
	tmp :	oscat_STRING250;
	a :	INT;
	b :	INT;
	c :	oscat_STRING1;
	stp :	INT;
END_VAR

(*@KEY@: WORKSHEET
NAME: REPLACE_CHARS
IEC_LANGUAGE: ST
*)
REPLACE_CHARS := STR;
(* make sure rep and src are of same length and length is > 0 *)
a := LEN(src);
b := LEN(rep);
IF a < b THEN
	rep := LEFT(rep, a);
ELSIF b < a THEN
	src := LEFT(src, b);
END_IF;

(* search the string and replace if necessary *)
stp := LEN(str);
FOR a := 1 TO stp DO
	c := MID(REPLACE_CHARS, 1, a);
	b := FIND(src, c);
	IF b > 0 THEN
        tmp := MID(rep, 1, b);
		REPLACE_CHARS := REPLACE(REPLACE_CHARS, tmp, 1, a);
	END_IF;
END_FOR;

(* revision history
hm		14. may. 2008	rev 1.0
	original version

*)
(*@KEY@: END_WORKSHEET *)
END_FUNCTION_BLOCK

(* ---- REPLACE_UML.ST ---- *)
(*@PROPERTIES_EX@
TYPE: POU
LOCALE: 0
IEC_LANGUAGE: ST
PLC_TYPE: independent
PROC_TYPE: independent
GROUP: STRINGS
*)
(*@KEY@:DESCRIPTION*)
version 1.1	29. mar. 2008
programmer 		kurt
tested by		hugo

REPLACE_UML replaces all occurences of Ä,Ö,Ü and ä,ö,ü,ß with Ae, ae, Oe, oe, Ue, ue and ss.
(*@KEY@:END_DESCRIPTION*)
FUNCTION_BLOCK REPLACE_UML

(*Group:Default*)

VAR_INPUT
	STR :	STRING;
END_VAR

VAR_OUTPUT
	REPLACE_UML :	STRING;
END_VAR

VAR
	pos1 :	INT;
	pos2 :	INT;
	l :	INT;
	pto :	BYTE;
	temp :	STRING;
	TO_UML :	TO_UML;
END_VAR

(*@KEY@: WORKSHEET
NAME: REPLACE_UML
IEC_LANGUAGE: ST
*)
L := LEN(str);
REPLACE_UML := str;
pos1 := 1;
pos2 := 1;
WHILE pos1 <= L AND pos2 <= 80 DO
    pto := INT_TO_BYTE(GET_CHAR(str,pos1));
	IF pto > BYTE#127 THEN
        TO_UML(IN:=pto);
        IF LEN(TO_UML.TO_UML) = 2 THEN
            temp := REPLACE_UML;
            IF pos2 >= 80 THEN
			     TO_UML.TO_UML := LEFT(TO_UML.TO_UML,1);
                 REPLACE_UML:=REPLACE(temp,TO_UML.TO_UML,1,pos2);
            ELSE
                 REPLACE_UML:=REPLACE(temp,TO_UML.TO_UML,1,pos2);
                 POS2 := POS2 +1;
            END_IF;
        END_IF;
    END_IF;
    pos1 := POS1 +1;
    pos2 := POS2 +1;
END_WHILE;

(* revision history
hm	29. feb 2008	rev 1.0
	original version

hm	29. mar. 2008	rev 1.1
	changed STRING to STRING(STRING_LENGTH)
	new code to avoid pointer out of range
	use new function to_uml
*)
(*@KEY@: END_WORKSHEET *)
END_FUNCTION_BLOCK

(* ---- RMP_B.ST ---- *)
(*@PROPERTIES_EX@
TYPE: POU
LOCALE: 0
IEC_LANGUAGE: ST
PLC_TYPE: independent
PROC_TYPE: independent
GROUP: ENGINEERING.SIGNAL_GENERATORS
*)
(*@KEY@:DESCRIPTION*)
version 2.0	23. oct. 2008
programmer 	oscat
tested BY	oscat

this ramp generator generates a byte wide ramp with 255 steps
the generator has an asynchronous set and reset
the ramp is controlled by PT which is the total ramp time for a full sweep from 0..255
an UD input controlls the direction Up or Down and the E input enables the ramp generation
a busy output indicates that the ramp is running, busy false means output is stable.
the outputs low and high will be true when the output has reached its max or min value.
(*@KEY@:END_DESCRIPTION*)
FUNCTION_BLOCK RMP_B

(*Group:Default*)

VAR_INPUT
	SET :	BOOL;
	PT :	TIME;
	E :	BOOL := TRUE;
	UP :	BOOL := TRUE;
	RST :	BOOL;
END_VAR

VAR_OUTPUT
	OUT :	BYTE;
	BUSY :	BOOL;
	HIGH :	BOOL;
	LOW :	BOOL;
END_VAR

VAR
	rmp :	_RMP_B;
END_VAR

(*@KEY@: WORKSHEET
NAME: RMP_B
IEC_LANGUAGE: ST
*)
(* generate ramp *)
rmp(dir := UP, E := E, TR := PT, RMP := out);
out := rmp.RMP;

(* set or reset operation *)
IF RST THEN
	out := BYTE#0;
ELSIF SET THEN
	out := BYTE#255;
END_IF;

(* checks for outputs stable and reset or set busy flag *)
low := out = BYTE#0;
high := out = BYTE#255;
busy := NOT (low OR high) AND E;

(* revision history

hm 5.10.2006	rev 1.1
	added busy output
hm 17.1.2007	rev 1.2
	renamed input ud to up for better usability
	deleted unused variable step

hm	17.9.2007		rev 1.3
	replaced time() with t_plc_ms() for compatibility reasons

hm	28. sep 2007	rev 1.4
	added outputs on and off
	busy is now disabled while en is false
	new coding for higher accuracy and performance

hm	5. oct 2007	rev 1.5
	added statements to allow for PT to be t#0s output jumps to max or min immediately

hm	25. dec 2007	rev 1.6
	improved code for better performance

hm	16. oct. 2008	rev 1.7
	improved code for better performance

hm	18. oct. 2008	rev 1.8
	added type conversion to avoid warnings
	changed input en to e for compatibility reasons

hm	23. oct. 2008	REV 	2.0
	new code using _RMP_B

*)
(*@KEY@: END_WORKSHEET *)
END_FUNCTION_BLOCK

(* ---- RMP_SOFT.ST ---- *)
(*@PROPERTIES_EX@
TYPE: POU
LOCALE: 0
IEC_LANGUAGE: ST
PLC_TYPE: independent
PROC_TYPE: independent
GROUP: ENGINEERING.SIGNAL_GENERATORS
*)
(*@KEY@:DESCRIPTION*)
version 2.0	26. oct. 2008
programmer 	oscat
tested BY	oscat

this soft on/off ramp generator generates a soft on and soft off ramp while the max on value is set by the input
the time for a full ramp can be set by config variables for up and down ramp.
(*@KEY@:END_DESCRIPTION*)
FUNCTION_BLOCK RMP_SOFT

(*Group:Default*)

VAR_INPUT
	IN :	BOOL;
	VAL :	BYTE;
	PT_ON :	TIME := T#100ms;
	PT_OFF :	TIME := T#100ms;
END_VAR

VAR_OUTPUT
	OUT :	BYTE := BYTE#00;
END_VAR

VAR
	rmp :	_RMP_B;
	tmp :	BYTE;
END_VAR

(*@KEY@: WORKSHEET
NAME: RMP_SOFT
IEC_LANGUAGE: ST
*)
tmp := SEL(in, BYTE#0, val);
IF tmp > out THEN
	(* we need to ramp down *)
	rmp(dir := TRUE, E := TRUE, TR := PT_ON, RMP := out);
	out := rmp.RMP;
	(* make sure out does not surpass tmp *)
	out := MIN(out, tmp);
ELSIF tmp < out THEN
	(* we need to ramp up *)
	rmp(dir := FALSE, E := TRUE, TR := PT_OFF, RMP := out);
	out := rmp.RMP;
	(* make sure out does not surpass tmp *)
	out := MAX(out, tmp);
ELSE
	(* no ramp necessary *)
	rmp(E := FALSE, RMP := out);
	out := rmp.RMP;
END_IF;

(* revision history

hm 22.1.2007	rev 1.1
	deleted unused variables X1 and I, X2 and X3

hm	17.9.2007	rev 1.2
	replaced time() with t_plc_ms() for compatibility reasons

hm	26. oct. 2008	2.0
	new code using _rmp_b
*)
(*@KEY@: END_WORKSHEET *)
END_FUNCTION_BLOCK

(* ---- RMP_W.ST ---- *)
(*@PROPERTIES_EX@
TYPE: POU
LOCALE: 0
IEC_LANGUAGE: ST
PLC_TYPE: independent
PROC_TYPE: independent
GROUP: ENGINEERING.SIGNAL_GENERATORS
*)
(*@KEY@:DESCRIPTION*)
version 2.0	23. oct. 2008
programmer 	oscat
tested BY	oscat

this ramp generator generates a Word wide ramp with 65535 steps
the generator has an asynchronous set and reset
the ramp is controlled by PT which is the total ramp time for a full sweep from 0..65535
an UD input controlls the direction Up or Down and the E input enables the ramp generation
a busy output indicates that the ramp is running, busy false means output is stable.
the outputs low and high will be true when the output has reached its max or min value.
(*@KEY@:END_DESCRIPTION*)
FUNCTION_BLOCK RMP_W

(*Group:Default*)

VAR_INPUT
	SET :	BOOL;
	PT :	TIME;
	E :	BOOL := TRUE;
	UP :	BOOL := TRUE;
	RST :	BOOL;
END_VAR

VAR_OUTPUT
	OUT :	WORD;
	BUSY :	BOOL;
	HIGH :	BOOL;
	LOW :	BOOL;
END_VAR

VAR
	rmp :	_RMP_W;
END_VAR

(*@KEY@: WORKSHEET
NAME: RMP_W
IEC_LANGUAGE: ST
*)
(* generate ramp *)
rmp(dir := UP, E := E, TR := PT, rmp := out);
out := rmp.RMP;

(* set or reset operation *)
IF RST THEN
	out := WORD#0;
ELSIF SET THEN
	out := WORD#65535;
END_IF;

(* checks for outputs stable and reset or set busy flag *)
low := out = WORD#0;
high := out = WORD#65535;
busy := NOT (low OR high) AND E;

(* revision history:

hm 4.10.2006		rev 1.1
	added the busy output which signals that the ramp is running.

hm 22.1.2007		rev 1.2
	deleted unused variable step

hm	17.9.2007		rev 1.3
	replaced time() with t_plc_ms() for compatibility reasons

hm	28. sep 2007	rev 1.4
	added outputs on and off
	busy is now disabled while en is false
	new coding for higher accuracy and performance

hm	5. oct 2007	rev 1.5
	added statements to allow for PT to be t#0s output jumps to max or min immediately

hm	2. dec 2007	rev 1.6
	corrected an error in calculation of step response

hm	25. dec 2007	rev 1.7
	corrected an error while step response was too slow for fast rise times

hm	16. oct. 2008	rev 1.8
	improved performance

hm	18. oct. 2008	rev 1.9
	renamed inout EN to E for compatibility reasons

hm	23. oct. 2008	rev 2.0
	new code using _RMP_W
*)
(*@KEY@: END_WORKSHEET *)
END_FUNCTION_BLOCK

(* ---- RTC_2.ST ---- *)
(*@PROPERTIES_EX@
TYPE: POU
LOCALE: 0
IEC_LANGUAGE: ST
PLC_TYPE: independent
PROC_TYPE: independent
GROUP: TIME_DATE
*)
(*@KEY@:DESCRIPTION*)
version 1.4	27.	apr. 2011
programmer 	hugo
tested by	tobias

RTC_2 is a real time clock module which runs utc and generates local time from utc.
daylight savings time can be enabled with den and an additional local time is generated with a delay of ofs im minutes.

(*@KEY@:END_DESCRIPTION*)
FUNCTION_BLOCK RTC_2

(*Group:Default*)

VAR_INPUT
	SET :	BOOL;
	SDT :	UDINT;
	SMS :	INT;
	DEN :	BOOL;
	OFS :	INT;
END_VAR

VAR_OUTPUT
	UDT :	UDINT;
	LDT :	UDINT;
	DSO :	BOOL;
	XMS :	INT;
END_VAR

VAR
	RT :	RTC_MS;
END_VAR

(*@KEY@: WORKSHEET
NAME: RTC_2
IEC_LANGUAGE: ST
*)
(* call rtc *)
RT(SET := SET, SDT := SDT, SMS := SMS);
UDT := rt.xdt;
XMS := rt.XMS;

(* check for daylight savings time and set dso output *)
dso := DST(udt) AND DEN;

(* calculate time offset and set ldt output *)
LDT := UDT + _INT_TO_UDINT(ofs + BOOL_TO_INT(DSO) * 60) * UDINT#60;

(* revision history
hm		20. jan. 2008	rev 1.0
	original version

hm		20. feb. 2008	rev 1.1
	added Millisecond Set input

hm		12. jun. 2008	rev 1.2
	improved performance

hm		20. jan. 2011	rev 1.3
	changed offset to be in minutes

hm		27. apr. 2011	rev 1.4
	fixed error with local time calculation

*)

(*@KEY@: END_WORKSHEET *)
END_FUNCTION_BLOCK

(* ---- RTC_MS.ST ---- *)
(*@PROPERTIES_EX@
TYPE: POU
LOCALE: 0
IEC_LANGUAGE: ST
PLC_TYPE: independent
PROC_TYPE: independent
GROUP: TIME_DATE
*)
(*@KEY@:DESCRIPTION*)
version 1.1	20. feb. 2008
programmer 	hugo
tested by	tobias

RTC_MS is a real time clock module which can be set to SDT when set is TRUE and the outputs XDT and XT present the DateTime and TOD with a resolution of milliseconds.
(*@KEY@:END_DESCRIPTION*)
FUNCTION_BLOCK RTC_MS

(*Group:Default*)

VAR_INPUT
	SET :	BOOL;
	SDT :	UDINT;
	SMS :	INT;
END_VAR

VAR_OUTPUT
	XDT :	UDINT;
	XMS :	INT;
END_VAR

VAR
	init :	BOOL;
	last :	UDINT;
	tx :	UDINT;
	T_PLC_MS :	T_PLC_MS;
END_VAR

(*@KEY@: WORKSHEET
NAME: RTC_MS
IEC_LANGUAGE: ST
*)
(* read system time *)
T_PLC_MS();
tx:= T_PLC_MS.T_PLC_MS;

IF set OR NOT init THEN
	(* clock needs to be set when set is true or after power up *)
	init := TRUE;
	xdt := SDT;
	XMS := SMS;
ELSE
	XMS := XMS + UDINT_TO_INT(tx - last);
	(* check if one second has expired *)
	IF XMS > 999 THEN
		XDT := XDT + UDINT#1; (* add one second *)
		XMS := XMS - 1000;
	END_IF;
END_IF;
last := tx;

(* revision history
hm		20. jan. 2008	rev 1.0
	original version

hm		20. feb. 2008	rev 1.1
	added Millisecond Set input
*)
(*@KEY@: END_WORKSHEET *)
END_FUNCTION_BLOCK

(* ---- SCHEDULER.ST ---- *)
(*@PROPERTIES_EX@
TYPE: POU
LOCALE: 0
IEC_LANGUAGE: ST
PLC_TYPE: independent
PROC_TYPE: independent
GROUP: LOGIC.GENERATORS
*)
(*@KEY@:DESCRIPTION*)
version 1.0	28. sep 2008
programmer 	hugo
tested by	tobias

SCHEDULER is used to call programs or function blocks at specific intervals.
T0..T3 defines the interval times.
(*@KEY@:END_DESCRIPTION*)
FUNCTION_BLOCK SCHEDULER

(*Group:Default*)

VAR_INPUT
	E0 :	BOOL;
	E1 :	BOOL;
	E2 :	BOOL;
	E3 :	BOOL;
	T0 :	TIME;
	T1 :	TIME;
	T2 :	TIME;
	T3 :	TIME;
END_VAR

VAR_OUTPUT
	Q0 :	BOOL;
	Q1 :	BOOL;
	Q2 :	BOOL;
	Q3 :	BOOL;
END_VAR

VAR
	T_PLC_MS :	T_PLC_MS;
	init :	BOOL;
	s0 :	TIME;
	s1 :	TIME;
	s2 :	TIME;
	s3 :	TIME;
	tx :	TIME;
	c :	INT;
END_VAR

(*@KEY@: WORKSHEET
NAME: SCHEDULER
IEC_LANGUAGE: ST
*)
(* read sps timer *)
T_PLC_MS();
tx:= UDINT_TO_TIME(T_PLC_MS.T_PLC_MS);

IF NOT init THEN
	init := TRUE;
	s0 := tx - T0;
	s1 := tx - T1;
	s2 := tx - T2;
	s3 := tx - T3;
END_IF;

Q0 := FALSE;
Q1 := FALSE;
Q2 := FALSE;
Q3 := FALSE;

CASE c OF
	0: 	IF tx - s0 >= T0 THEN
			Q0 := E0;
			s0 := tx;
		END_IF;
		c := 1;
	1: 	IF tx - s1 >= T1 THEN
			Q1 := E1;
			s1 := tx;
		END_IF;
		c := 2;
	2: 	IF tx - s2 >= T2 THEN
			Q2 := E2;
			s2 := tx;
		END_IF;
		c := 3;
	3: 	IF tx - s3 >= T3 THEN
			Q3 := E3;
			s3 := tx;
		END_IF;
		c := 0;
END_CASE;

(* revision history

hm 28. sep. 2008		rev 1.0
	original version

*)
(*@KEY@: END_WORKSHEET *)
END_FUNCTION_BLOCK

(* ---- SCHEDULER_2.ST ---- *)
(*@PROPERTIES_EX@
TYPE: POU
LOCALE: 0
IEC_LANGUAGE: ST
PLC_TYPE: independent
PROC_TYPE: independent
GROUP: LOGIC.GENERATORS
*)
(*@KEY@:DESCRIPTION*)
version 1.0	29. sep 2008
programmer 	hugo
tested by	tobias

SCHEDULER_2 is used to call programs or function blocks at specific cycles.
C0..C3 defines after how many cycles the output becomes active.
O0..O3 defines a cycle offset at startup.
(*@KEY@:END_DESCRIPTION*)
FUNCTION_BLOCK SCHEDULER_2

(*Group:Default*)

VAR_INPUT
	E0 :	BOOL;
	E1 :	BOOL;
	E2 :	BOOL;
	E3 :	BOOL;
	C0 :	UINT;
	C1 :	UINT;
	C2 :	UINT;
	C3 :	UINT;
	O0 :	UINT;
	O1 :	UINT;
	O2 :	UINT;
	O3 :	UINT;
END_VAR

VAR_OUTPUT
	Q0 :	BOOL;
	Q1 :	BOOL;
	Q2 :	BOOL;
	Q3 :	BOOL;
END_VAR

VAR
	sx :	UINT;
END_VAR

(*@KEY@: WORKSHEET
NAME: SCHEDULER_2
IEC_LANGUAGE: ST
*)
Q0 := E0 AND (sx MOD C0 - O0 = UINT#0);
Q1 := E1 AND (sx MOD C1 - O1 = UINT#0);
Q2 := E2 AND (sx MOD C2 - O2 = UINT#0);
Q3 := E3 AND (sx MOD C3 - O3 = UINT#0);

(* increment cycle counter every cycle *)
sx := sx + UINT#1;

(* revision history
hm 29. sep. 2008		rev 1.0
	original version

*)
(*@KEY@: END_WORKSHEET *)
END_FUNCTION_BLOCK

(* ---- SDT_TO_DATE.ST ---- *)
(*@PROPERTIES_EX@
TYPE: POU
LOCALE: 0
IEC_LANGUAGE: ST
PLC_TYPE: independent
PROC_TYPE: independent
GROUP: TIME_DATE
*)
(*@KEY@:DESCRIPTION*)
version 1.0	18. oct 2008
programmer 	hugo
tested by	oscat

converts Structured date time (SDT) to Date Time
(*@KEY@:END_DESCRIPTION*)
FUNCTION_BLOCK SDT_TO_DATE

(*Group:Default*)

VAR_INPUT
	DTI :	oscat_SDT;
END_VAR

VAR_OUTPUT
	SDT_TO_DATE :	UDINT;
END_VAR

(*@KEY@: WORKSHEET
NAME: SDT_TO_DATE
IEC_LANGUAGE: ST
*)
SDT_TO_DATE := SET_DATE(DTI.YEAR, DTI.MONTH, DTI.DAY);

(* revision history

hm 18. oct. 2008	rev 1.0
	original version

*)
(*@KEY@: END_WORKSHEET *)
END_FUNCTION_BLOCK

(* ---- SDT_TO_DT.ST ---- *)
(*@PROPERTIES_EX@
TYPE: POU
LOCALE: 0
IEC_LANGUAGE: ST
PLC_TYPE: independent
PROC_TYPE: independent
GROUP: TIME_DATE
*)
(*@KEY@:DESCRIPTION*)
version 1.0	18. oct 2008
programmer 	hugo
tested by	oscat

converts Structured date time (SDT) to Date Time
(*@KEY@:END_DESCRIPTION*)
FUNCTION_BLOCK SDT_TO_DT

(*Group:Default*)

VAR_INPUT
	DTI :	oscat_SDT;
END_VAR

VAR_OUTPUT
	SDT_TO_DT :	UDINT;
END_VAR

(*@KEY@: WORKSHEET
NAME: SDT_TO_DT
IEC_LANGUAGE: ST
*)
SDT_TO_DT := SET_DT(DTI.YEAR, DTI.MONTH, DTI.DAY, DTI.HOUR, DTI.MINUTE, DTI.SECOND);

(* revision history

hm 18. oct. 2008	rev 1.0
	original version

*)
(*@KEY@: END_WORKSHEET *)
END_FUNCTION_BLOCK

(* ---- SDT_TO_TOD.ST ---- *)
(*@PROPERTIES_EX@
TYPE: POU
LOCALE: 0
IEC_LANGUAGE: ST
PLC_TYPE: independent
PROC_TYPE: independent
GROUP: TIME_DATE
*)
(*@KEY@:DESCRIPTION*)
version 1.0	18. oct 2008
programmer 	hugo
tested by	oscat

converts Structured date time (SDT) to Date Time
(*@KEY@:END_DESCRIPTION*)
FUNCTION_BLOCK SDT_TO_TOD

(*Group:Default*)

VAR_INPUT
	DTI :	oscat_SDT;
END_VAR

VAR_OUTPUT
	SDT_TO_TOD :	UDINT;
END_VAR

(*@KEY@: WORKSHEET
NAME: SDT_TO_TOD
IEC_LANGUAGE: ST
*)
SDT_TO_TOD := _INT_TO_UDINT(DTI.HOUR) * UDINT#3600000 + _INT_TO_UDINT(DTI.MINUTE) * UDINT#60000 + _INT_TO_UDINT(DTI.SECOND) * UDINT#1000 + _INT_TO_UDINT(DTI.MS);

(* revision history

hm 18. oct. 2008	rev 1.0
	original version

*)
(*@KEY@: END_WORKSHEET *)
END_FUNCTION_BLOCK

(* ---- SEL2_OF_3.ST ---- *)
(*@PROPERTIES_EX@
TYPE: POU
LOCALE: 0
IEC_LANGUAGE: ST
PLC_TYPE: independent
PROC_TYPE: independent
GROUP: ENGINEERING.SIGNAL_PROCESSING
*)
(*@KEY@:DESCRIPTION*)
version 1.1	10. mar. 2009
programmer 	oscat
tested BY	oscat

SEL2_OF_3 checks if 3 input Signals are within a distance D from each other and calculates the average of the 3 inputs do not offset more than D from each other.
If 1 input is more than D greater or smaller than any other input it will be ignored and the average will be calcualted from the remaining 2 Inputs.
In the case the Output is only calculated from 2 Inputs a Warning Output W will display the Number of the discarded Input. if none of the 3 Inputs are within the allowed Delata D from each other,
an Error Output E is set True and the last valid Output will remain active until at least 2 Inputs are within a valid Range from each other.

(*@KEY@:END_DESCRIPTION*)
FUNCTION_BLOCK SEL2_OF_3

(*Group:Default*)

VAR_INPUT
	IN1 :	REAL;
	IN2 :	REAL;
	IN3 :	REAL;
	D :	REAL;
END_VAR

VAR_OUTPUT
	Y :	REAL;
	W :	INT;
	E :	BOOL;
END_VAR

VAR
	D12 :	BOOL;
	D23 :	BOOL;
	D31 :	BOOL;
END_VAR

(*@KEY@: WORKSHEET
NAME: SEL2_OF_3
IEC_LANGUAGE: ST
*)
D12 := ABS(IN1-IN2) <= D;
D23 := ABS(IN2-IN3) <= D;
D31 := ABS(IN3-IN1) <= D;

IF (D12 AND D23) OR (D12 AND D31) OR (D23 AND D31) THEN
	(* all 3 inputs are valid *)
	Y := (IN1 + IN2 + IN3) * 0.333333333333;
	E := FALSE;
	W := 0;
ELSIF D12 THEN
	(* only inut 1 and 2 are valid *)
	Y := (In1 + IN2) * 0.5;
	E := FALSE;
	W := 3;
ELSIF D23 THEN
	(* only inut 2 and 3 are valid *)
	Y := (In2 + IN3) * 0.5;
	E := FALSE;
	W := 1;
ELSIF D31 THEN
	(* only inut 3 and 1 are valid *)
	Y := (In3 + IN1) * 0.5;
	E := FALSE;
	W := 2;
ELSE
	(* no calculation possible *)
	E := TRUE;
	W := 4;
END_IF;

(* revision history
hm	18. may 2008	rev 1.0
	original version

hm	10. mar. 2009	rev 1.1
	improved code
*)
(*@KEY@: END_WORKSHEET *)
END_FUNCTION_BLOCK

(* ---- SEL2_OF_3B.ST ---- *)
(*@PROPERTIES_EX@
TYPE: POU
LOCALE: 0
IEC_LANGUAGE: ST
PLC_TYPE: independent
PROC_TYPE: independent
GROUP: ENGINEERING.SIGNAL_PROCESSING
*)
(*@KEY@:DESCRIPTION*)
version 1.0	19. may. 2008
programmer 	oscat
tested BY	oscat

SEL2_OF_3B is used to connect 3 binary sensors to one signal. the output Q reflects the state of at least two inputs.
if two or more of the 3 inputs ate TRUE then Q will be TRUE and if two or more of the three inputs are FALSE then Q will be false.
the main putrpose is the connection of 3 redundant binary sensors.
The output W will be active when one of the 3 inputs is of different state.
to avoid flickering while the sensors are switching the output W will become active after a programmed delay of TD.
(*@KEY@:END_DESCRIPTION*)
FUNCTION_BLOCK SEL2_OF_3B

(*Group:Default*)

VAR_INPUT
	IN1 :	BOOL;
	IN2 :	BOOL;
	IN3 :	BOOL;
	TD :	TIME;
END_VAR

VAR_OUTPUT
	Q :	BOOL;
	W :	BOOL;
END_VAR

VAR
	TDEL :	TON;
END_VAR

(*@KEY@: WORKSHEET
NAME: SEL2_OF_3B
IEC_LANGUAGE: ST
*)
Q := (IN1 AND IN2) OR (IN1 AND IN3) OR (IN2 AND IN3);
TDEL(IN := (in1 XOR in2) OR (in1 XOR in3) OR (in2 XOR in3), PT := TD);
W := TDEL.Q;

(* revision history
hm		19. may 2008	rev 1.0
	original version

*)
(*@KEY@: END_WORKSHEET *)
END_FUNCTION_BLOCK

(* ---- SELECT_8.ST ---- *)
(*@PROPERTIES_EX@
TYPE: POU
LOCALE: 0
IEC_LANGUAGE: ST
PLC_TYPE: independent
PROC_TYPE: independent
GROUP: LOGIC.FF_EDGE_TRIGGERED
*)
(*@KEY@:DESCRIPTION*)
version 1.1	27. feb. 2009
programmer 	hugo
tested BY	tobias

select_8 selects one of 8 outputs at any time. the outputscan be selected by up or down keys and an independent anable switches all outouts off if set false
(*@KEY@:END_DESCRIPTION*)
FUNCTION_BLOCK SELECT_8

(*Group:Default*)

VAR_INPUT
	E :	BOOL;
	SET :	BOOL;
	IN :	BYTE;
	UP :	BOOL;
	DN :	BOOL;
	RST :	BOOL;
END_VAR

VAR_OUTPUT
	Q0 :	BOOL;
	Q1 :	BOOL;
	Q2 :	BOOL;
	Q3 :	BOOL;
	Q4 :	BOOL;
	Q5 :	BOOL;
	Q6 :	BOOL;
	Q7 :	BOOL;
	STATE :	INT;
END_VAR

VAR
	last_up :	BOOL;
	last_dn :	BOOL;
END_VAR

(*@KEY@: WORKSHEET
NAME: SELECT_8
IEC_LANGUAGE: ST
*)
IF rst THEN
	state := 0;
ELSIF set THEN
	state := _BYTE_TO_INT(IN);
ELSIF up AND NOT last_up THEN
	state := inc(state,1,7);
ELSIF dn AND NOT last_dn THEN
	state := inc(state,-1,7);
END_IF;
last_UP := UP;
last_DN := DN;

Q0 := FALSE;
Q1 := FALSE;
Q2 := FALSE;
Q3 := FALSE;
Q4 := FALSE;
Q5 := FALSE;
Q6 := FALSE;
Q7 := FALSE;

IF e THEN
	CASE state OF
		0: Q0 := TRUE;
		1: Q1 := TRUE;
		2: Q2 := TRUE;
		3: Q3 := TRUE;
		4: Q4 := TRUE;
		5: Q5 := TRUE;
		6: Q6 := TRUE;
		7: Q7 := TRUE;
	END_CASE;
END_IF;

(* revision history
hm	16. jan 2008	rev 1.0
	original version

*)
(*@KEY@: END_WORKSHEET *)
END_FUNCTION_BLOCK

(* ---- SEQUENCE_4.ST ---- *)
(*@PROPERTIES_EX@
TYPE: POU
LOCALE: 0
IEC_LANGUAGE: ST
PLC_TYPE: independent
PROC_TYPE: independent
GROUP: LOGIC.GENERATORS
*)
(*@KEY@:DESCRIPTION*)
version 1.4	17 sep 2007
programmer 	oscat
tested by	hans

sequence_4 enables run when a low to high transition is present on start.
a low to high transition on start will restart the sequencer at any time while a rst will hold the sequencer in reset while true.
after run is enabled with a rising edge on start the sequencer waits for wait0 on in0 to enable q0 which stays on for delay0.
the next cycle starts with wait1, continues with delay 1 and so on...
if an edge is not detected during the wait period, the sequencer will then display the error number on the status output.
the status numbers 1..4 are errors in step 0..3.
after the last step that sets q3, the sequencer leaves q3 on for delay3 and then resets to the initial state.
a step output will indicate the current step of the sequencer and will also be present with a fault condition.
after the first output is turened on the sequencer switches from q0 to q1 and so on, at any time there is only one output enabled.
if an input signal is not detected during a wait period, the sequencer will display the error number ( 1 for in0, 2 for in1 .... ).
when an error is present and the config variable stop_on_error is set then the sequencer will stop. otherwise it will continue.
The status output will also display 110 for waiting and 111 for sequence running.

(*@KEY@:END_DESCRIPTION*)
FUNCTION_BLOCK SEQUENCE_4

(*Group:Default*)

VAR_INPUT
	IN0 :	BOOL := TRUE;
	IN1 :	BOOL := TRUE;
	IN2 :	BOOL := TRUE;
	IN3 :	BOOL := TRUE;
	START :	BOOL;
	RST :	BOOL;
	WAIT0 :	TIME;
	DELAY0 :	TIME;
	WAIT1 :	TIME;
	DELAY1 :	TIME;
	WAIT2 :	TIME;
	DELAY2 :	TIME;
	WAIT3 :	TIME;
	DELAY3 :	TIME;
	STOP_ON_ERROR :	BOOL;
END_VAR

VAR_OUTPUT
	Q0 :	BOOL;
	Q1 :	BOOL;
	Q2 :	BOOL;
	Q3 :	BOOL;
	QX :	BOOL;
	RUN :	BOOL;
	STEP :	INT := -1;
	STATUS :	BYTE;
END_VAR

VAR
	last :	TIME;
	edge :	BOOL;
	tx :	TIME;
	init :	BOOL;
	T_PLC_MS :	T_PLC_MS;
END_VAR

(*@KEY@: WORKSHEET
NAME: SEQUENCE_4
IEC_LANGUAGE: ST
*)
(* read sps timer *)
T_PLC_MS();
tx:= UDINT_TO_TIME(T_PLC_MS.T_PLC_MS);

(* initialize on startup *)
IF NOT init THEN
	last := tx;
	init := TRUE;
	status := BYTE#110;
END_IF;

(* asynchronous reset *)
IF rst THEN
	step := -1;
	Q0 := FALSE;
	Q1 := FALSE;
	Q2 := FALSE;
	Q3 := FALSE;
	status := BYTE#110;
	run := FALSE;

(* edge on start input restarts the sequencer *)
ELSIF start AND NOT edge THEN
	step := 0;
	last := tx;
	status := BYTE#111;
	Q0 := FALSE;
	Q1 := FALSE;
	Q2 := FALSE;
	Q3 := FALSE;
	run := TRUE;
END_IF;
edge := start;

(* check if stop on status is necessary *)
IF status > BYTE#0 AND status < BYTE#100 AND stop_on_error THEN RETURN; END_IF;

(* sequence is running *)
IF run AND step = 0 THEN
	IF NOT q0 AND in0 AND tx - last <= wait0 THEN
		Q0 := TRUE;
		last := tx;
	ELSIF NOT q0 AND tx - last > wait0 THEN
		status := BYTE#1;
		run := FALSE;
	ELSIF q0 AND tx - last >= delay0 THEN
		step := 1;
		last := tx;
	END_IF;
END_IF;
IF run AND step = 1 THEN
	IF NOT q1 AND in1 AND tx - last <= wait1 THEN
		Q0 := FALSE;
		Q1 := TRUE;
		last := tx;
	ELSIF NOT q1 AND Tx - last > wait1 THEN
		status := BYTE#2;
		q0 := FALSE;
		run := FALSE;
	ELSIF q1 AND tx - last >= delay1 THEN
		step := 2;
		last := tx;
	END_IF;
END_IF;
IF run AND step = 2 THEN
	IF NOT q2 AND in2 AND tx - last <= wait2 THEN
		Q1 := FALSE;
		Q2 := TRUE;
		last := tx;
	ELSIF NOT q2 AND Tx - last > wait2 THEN
		status := BYTE#3;
		q1 := FALSE;
		run := FALSE;
	ELSIF q2 AND tx - last >= delay2 THEN
		step := 3;
		last := tx;
	END_IF;
END_IF;
IF run AND step = 3 THEN
	IF NOT q3 AND in3 AND tx - last <= wait3 THEN
		Q2 := FALSE;
		Q3 := TRUE;
		last := tx;
	ELSIF NOT q3 AND Tx - last > wait3 THEN
		status := BYTE#4;
		q2 := FALSE;
		run := FALSE;
	ELSIF q3 AND tx - last >= delay3 THEN
		step := -1;
		q3 := FALSE;
		run := FALSE;
		status := BYTE#110;
	END_IF;
END_IF;
QX := q0 OR q1 OR q2 OR q3;

(*
hm 1.10.06		rev 1.1
	corrected delay logic to be after event and not before
	added any output

hm 1.12.06		rev 1.2
	corrected failure in sequence logic.
	added init at startup to prevent from initial error after start.

hm 17.1.2007		rev 1.3
	changed output fault to status for better compatibility with other modules (ESR).
	added stop on error functionality and setup variable
	default for inputs in0..3 is true.
	renamed variable state to step

hm	17.sep 2007		rev 1.4
	replaced time() with T_PLC_MS() for compatibility reasons

*)
(*@KEY@: END_WORKSHEET *)
END_FUNCTION_BLOCK

(* ---- SEQUENCE_64.ST ---- *)
(*@PROPERTIES_EX@
TYPE: POU
LOCALE: 0
IEC_LANGUAGE: ST
PLC_TYPE: independent
PROC_TYPE: independent
GROUP: LOGIC.GENERATORS
*)
(*@KEY@:DESCRIPTION*)
version 1.0	29. jun. 2008
programmer 	hugo
tested by	oscat

sequence generates a sequence of states with a programmable length for each state.
(*@KEY@:END_DESCRIPTION*)
FUNCTION_BLOCK SEQUENCE_64

(*Group:Default*)

VAR_INPUT
	START :	BOOL;
	SMAX :	INT;
	RST :	BOOL;
END_VAR

VAR_OUTPUT
	STATE :	INT := INT#-1;
	TRIG :	BOOL;
END_VAR

VAR_IN_OUT
	PROG :	oscat_array64_time;
END_VAR

VAR
	T_PLC_MS :	T_PLC_MS;
	tx :	TIME;
	last :	TIME;
	edge :	BOOL;
END_VAR

(*@KEY@: WORKSHEET
NAME: SEQUENCE_64
IEC_LANGUAGE: ST
*)
(* read system timer *)
T_PLC_MS();
tx:= UDINT_TO_TIME(T_PLC_MS.T_PLC_MS);
TRIG := FALSE;

IF RST THEN
	STATE := -1;

(* start sequence *)
ELSIF START AND NOT edge THEN
	STATE := 0;
	last := tx;
	TRIG := TRUE;

(* sequence generator *)
ELSIF (STATE >= 0) THEN
	IF (tx - last) >= PROG[STATE] THEN
		STATE := INC2(STATE, 1, -1, SMAX);
		last := tx;
		TRIG := TRUE;
	END_IF;
END_IF;

edge := START;

(* revision history
hm	29. jun. 2008
	original version

*)
(*@KEY@: END_WORKSHEET *)
END_FUNCTION_BLOCK

(* ---- SEQUENCE_8.ST ---- *)
(*@PROPERTIES_EX@
TYPE: POU
LOCALE: 0
IEC_LANGUAGE: ST
PLC_TYPE: independent
PROC_TYPE: independent
GROUP: LOGIC.GENERATORS
*)
(*@KEY@:DESCRIPTION*)
version 1.4	17 sep 2007
programmer 	oscat
tested by		hans

sequence_8 enables run when a low to high transition is present on start.
a low to high transition on start will restart the sequencer at any time while a rst will hold the sequencer in reset while true.
after run is enabled with a rising edge on start the sequencer waits for wait0 on in0 to enable q0 which stays on for delay0.
the next cycle starts with wait1, continues with delay 1 and so on...
if an edge is not detected during the wait period, the sequencer will then display the error number on the status output.
The status numbers are 1 .. 8 for erros in step 0..7.
after the last step that sets q7, the sequencer leaves q7 on for delay7 and then resets to the initial state.
a step output will indicate the current step of the sequencer and will also be present with a fault condition.
after the first output is turened on the sequencer switches from q0 to q1 and so on, at any time there is only one output enabled.
if an input signal is not detected during a wait period, the sequencer will display the error number ( 1 for in0, 2 for in1 .... ).
when an error is present and the config variable stop_on_error is set then the sequencer will stop. otherwise it will continue.
The status output will also display 110 for waiting and 111 sequece running.
(*@KEY@:END_DESCRIPTION*)
FUNCTION_BLOCK SEQUENCE_8

(*Group:Default*)

VAR_INPUT
	IN0 :	BOOL := TRUE;
	IN1 :	BOOL := TRUE;
	IN2 :	BOOL := TRUE;
	IN3 :	BOOL := TRUE;
	IN4 :	BOOL := TRUE;
	IN5 :	BOOL := TRUE;
	IN6 :	BOOL := TRUE;
	IN7 :	BOOL := TRUE;
	START :	BOOL;
	RST :	BOOL;
	WAIT0 :	TIME;
	DELAY0 :	TIME;
	WAIT1 :	TIME;
	DELAY1 :	TIME;
	WAIT2 :	TIME;
	DELAY2 :	TIME;
	WAIT3 :	TIME;
	DELAY3 :	TIME;
	WAIT4 :	TIME;
	DELAY4 :	TIME;
	WAIT5 :	TIME;
	DELAY5 :	TIME;
	WAIT6 :	TIME;
	DELAY6 :	TIME;
	WAIT7 :	TIME;
	DELAY7 :	TIME;
	STOP_ON_ERROR :	BOOL;
END_VAR

VAR_OUTPUT
	Q0 :	BOOL;
	Q1 :	BOOL;
	Q2 :	BOOL;
	Q3 :	BOOL;
	Q4 :	BOOL;
	Q5 :	BOOL;
	Q6 :	BOOL;
	Q7 :	BOOL;
	QX :	BOOL;
	RUN :	BOOL;
	STEP :	INT := -1;
	STATUS :	BYTE;
END_VAR

VAR
	last :	TIME;
	edge :	BOOL;
	tx :	TIME;
	init :	BOOL;
	T_PLC_MS :	T_PLC_MS;
END_VAR

(*@KEY@: WORKSHEET
NAME: SEQUENCE_8
IEC_LANGUAGE: ST
*)
(* read sps timer *)
T_PLC_MS();
tx:= UDINT_TO_TIME(T_PLC_MS.T_PLC_MS);

(* initialize on startup *)
IF NOT init THEN
	last := tx;
	init := TRUE;
	status := BYTE#110;
END_IF;

(* asynchronous reset *)
IF rst THEN
	step := -1;
	Q0 := FALSE;
	Q1 := FALSE;
	Q2 := FALSE;
	Q3 := FALSE;
	Q4 := FALSE;
	Q5 := FALSE;
	Q6 := FALSE;
	Q7 := FALSE;
	status := BYTE#110;
	run := FALSE;

(* edge on start input restarts the sequencer *)
ELSIF start AND NOT edge THEN
	step := 0;
	last := tx;
	status := BYTE#111;
	Q0 := FALSE;
	Q1 := FALSE;
	Q2 := FALSE;
	Q3 := FALSE;
	Q4 := FALSE;
	Q5 := FALSE;
	Q6 := FALSE;
	Q7 := FALSE;
	run := TRUE;
END_IF;
edge := start;

(* check if stop on error is necessary *)
IF status > BYTE#0 AND status < BYTE#100 AND stop_on_error THEN RETURN; END_IF;

(* sequence is running *)
IF run AND step = 0 THEN
	IF NOT q0 AND in0 AND tx - last <= wait0 THEN
		Q0 := TRUE;
		last := tx;
	ELSIF NOT q0 AND tx - last > wait0 THEN
		status := BYTE#1;
		run := FALSE;
	ELSIF q0 AND tx - last >= delay0 THEN
		step := 1;
		last := tx;
	END_IF;
END_IF;
IF run AND step = 1 THEN
	IF NOT q1 AND in1 AND tx - last <= wait1 THEN
		Q0 := FALSE;
		Q1 := TRUE;
		last := tx;
	ELSIF NOT q1 AND Tx - last > wait1 THEN
		status := BYTE#2;
		q0 := FALSE;
		run := FALSE;
	ELSIF q1 AND tx - last >= delay1 THEN
		step := 2;
		last := tx;
	END_IF;
END_IF;
IF run AND step = 2 THEN
	IF NOT q2 AND in2 AND tx - last <= wait2 THEN
		Q1 := FALSE;
		Q2 := TRUE;
		last := tx;
	ELSIF NOT q2 AND Tx - last > wait2 THEN
		status := BYTE#3;
		q1 := FALSE;
		run := FALSE;
	ELSIF q2 AND tx - last >= delay2 THEN
		step := 3;
		last := tx;
	END_IF;
END_IF;
IF run AND step = 3 THEN
	IF NOT q3 AND in3 AND tx - last <= wait3 THEN
		Q2 := FALSE;
		Q3 := TRUE;
		last := tx;
	ELSIF NOT q3 AND Tx - last > wait3 THEN
		status := BYTE#4;
		q2 := FALSE;
		run := FALSE;
	ELSIF q3 AND tx - last >= delay3 THEN
		step := 4;
		last := tx;
	END_IF;
END_IF;
IF run AND step = 4 THEN
	IF NOT q4 AND in4 AND tx - last <= wait4 THEN
		Q3 := FALSE;
		Q4 := TRUE;
		last := tx;
	ELSIF NOT q4 AND Tx - last > wait4 THEN
		status := BYTE#5;
		q3 := FALSE;
		run := FALSE;
	ELSIF q4 AND tx - last >= delay4 THEN
		step := 5;
		last := tx;
	END_IF;
END_IF;
IF run AND step = 5 THEN
	IF NOT q5 AND in5 AND tx - last <= wait5 THEN
		Q4 := FALSE;
		Q5 := TRUE;
		last := tx;
	ELSIF NOT q5 AND Tx - last > wait5 THEN
		status := BYTE#6;
		q4 := FALSE;
		run := FALSE;
	ELSIF q5 AND tx - last >= delay5 THEN
		step := 6;
		last := tx;
	END_IF;
END_IF;
IF run AND step = 6 THEN
	IF NOT q6 AND in6 AND tx - last <= wait6 THEN
		Q5 := FALSE;
		Q6 := TRUE;
		last := tx;
	ELSIF NOT q6 AND Tx - last > wait6 THEN
		status := BYTE#7;
		q5 := FALSE;
		run := FALSE;
	ELSIF q6 AND tx - last >= delay6 THEN
		step := 7;
		last := tx;
	END_IF;
END_IF;
IF run AND step = 7 THEN
	IF NOT q7 AND in7 AND tx - last <= wait7 THEN
		Q6 := FALSE;
		Q7 := TRUE;
		last := tx;
	ELSIF NOT q7 AND Tx - last > wait7 THEN
		status := BYTE#8;
		q6 := FALSE;
		run := FALSE;
	ELSIF q7 AND tx - last >= delay7 THEN
		step := -1;
		Q7 := FALSE;
		Run := FALSE;
		status := BYTE#110;
	END_IF;
END_IF;
QX := q0 OR q1 OR q2 OR q3 OR q4 OR q5 OR q6 OR q7;

(*
hm 1.10.06		rev 1.1
	corrected delay logic to be after event and not before
	added any output

hm 1.12.06		rev 1.2
	corrected failure in sequence logic.
	added init at startup to prevent from initial statuss after start.

hm 17.1.2007		rev 1.3
	changed output fault to status for better compatibility with other modules (ESR)
	added stop on error functionality and setup variable
	default for inputs in0..7 is true.
	renames variable state to step

hm	17.sep 2007		rev 1.4
	replaced time() with T_PLC_MS() for compatibility reasons

*)
(*@KEY@: END_WORKSHEET *)
END_FUNCTION_BLOCK

(* ---- SETUP_CHARNAMES.ST ---- *)
(*@PROPERTIES_EX@
TYPE: POU
LOCALE: 0
IEC_LANGUAGE: ST
PLC_TYPE: independent
PROC_TYPE: independent
GROUP: SETUP
*)
(*@KEY@:DESCRIPTION*)

(*@KEY@:END_DESCRIPTION*)
FUNCTION_BLOCK SETUP_CHARNAMES

(*Group:Default*)

VAR_IN_OUT
	CHARNAMES :	oscat_CHARNAMES;
END_VAR

VAR
	init :	BOOL;
END_VAR

(*@KEY@: WORKSHEET
NAME: SETUP_CHARNAMES
IEC_LANGUAGE: ST
*)
(* Daten initialisieren *)
IF init THEN RETURN; END_IF;

init := TRUE;

CHARNAMES[01] := ';"&quot;&&amp;<&lt;>&gt;€&euro; &nbsp;¡&iexcl;¢&cent;£&pound;¤&curren;¥&yen;';
CHARNAMES[02] := ';¦&brvbar;§&sect;¨&uml;©&copy;ª&ordf;«&laquo;¬&not;­&shy;®&reg;¯&macr;°&deg;';
CHARNAMES[03] := ';±&plusmn;²&sup2;³&sup3;´&acute;µ&micro;¶&para;·&middot;¸&cedil;¹&sup1;º&ordm;';
CHARNAMES[04] := ';»&raquo;¼&frac14;½&frac12;¾&frac34;¿&iquest;À&Agrave;Á&Aacute;Â&Acirc;Ã&Atilde;';
CHARNAMES[05] := ';Ä&Auml;Å&Aring;Æ&AElig;Ç&Ccedil;È&Egrave;É&Eacute;Ê&Ecirc;Ë&Euml;Ì&Igrave;';
CHARNAMES[06] := ';Í&Iacute;Î&Icirc;Ï&Iuml;Ð&ETH;Ñ&Ntilde;Ò&Ograve;Ó&Oacute;Ô&Ocirc;Õ&Otilde;';
CHARNAMES[07] := ';Ö&Ouml;×&times;Ø&Oslash;Ù&Ugrave;Ú&Uacute;Û&Ucirc;Ü&Uuml;Ý&Yacute;Þ&THORN;';
CHARNAMES[08] := ';ß&szlig;à&agrave;á&aacute;â&acirc;ã&atilde;ä&auml;å&aring;æ&aelig;ç&ccedil;';
CHARNAMES[09] := ';è&egrave;é&eacute;ê&ecirc;ë&euml;ì&igrave;í&iacute;î&icirc;ï&iuml;ð&eth;';
CHARNAMES[10] := ';ñ&ntilde;ò&ograve;ó&oacute;ô&ocirc;õ&otilde;ö&ouml;÷&divide;ø&oslash;ù&ugrave;';
CHARNAMES[11] := ';ú&uacute;û&ucirc;ü&uuml;ý&yacute;þ&thorn;ÿ&yuml;';
(*@KEY@: END_WORKSHEET *)
END_FUNCTION_BLOCK

(* ---- SETUP_DIRS.ST ---- *)
(*@PROPERTIES_EX@
TYPE: POU
LOCALE: 0
IEC_LANGUAGE: ST
PLC_TYPE: independent
PROC_TYPE: independent
GROUP: SETUP
*)
(*@KEY@:DESCRIPTION*)

(*@KEY@:END_DESCRIPTION*)
FUNCTION_BLOCK SETUP_DIRS

(*Group:Default*)

VAR_IN_OUT
	DIRS :	oscat_DIRS;
END_VAR

VAR
	init :	BOOL;
END_VAR

(*@KEY@: WORKSHEET
NAME: SETUP_DIRS
IEC_LANGUAGE: ST
*)
(* Daten initialisieren *)
IF init THEN RETURN; END_IF;
init := TRUE;

(* ---- english --- *)
DIRS[1][00] := 'N';
DIRS[1][01] := 'NNE';
DIRS[1][02] := 'NE';
DIRS[1][03] := 'ENE';
DIRS[1][04] := 'E';
DIRS[1][05] := 'ESE';
DIRS[1][06] := 'SE';
DIRS[1][07] := 'SSE';
DIRS[1][08] := 'S';
DIRS[1][09] := 'SSW';
DIRS[1][10] := 'SW';
DIRS[1][11] := 'WSW';
DIRS[1][12] := 'W';
DIRS[1][13] := 'WNW';
DIRS[1][14] := 'NW';
DIRS[1][15] := 'NNW';

(* ---- german --- *)
DIRS[2][00] := 'N';
DIRS[2][01] := 'NNO';
DIRS[2][02] := 'NO';
DIRS[2][03] := 'ONO';
DIRS[2][04] := 'O';
DIRS[2][05] := 'OSO';
DIRS[2][06] := 'SO';
DIRS[2][07] := 'SSO';
DIRS[2][08] := 'S';
DIRS[2][09] := 'SSW';
DIRS[2][10] := 'SW';
DIRS[2][11] := 'WSW';
DIRS[2][12] := 'W';
DIRS[2][13] := 'WNW';
DIRS[2][14] := 'NW';
DIRS[2][15] := 'NNW';

(* ---- french --- *)
DIRS[3][00] := 'N';
DIRS[3][01] := 'NNO';
DIRS[3][02] := 'NO';
DIRS[3][03] := 'ONO';
DIRS[3][04] := 'O';
DIRS[3][05] := 'OSO';
DIRS[3][06] := 'SO';
DIRS[3][07] := 'SSO';
DIRS[3][08] := 'S';
DIRS[3][09] := 'SSW';
DIRS[3][10] := 'SW';
DIRS[3][11] := 'WSW';
DIRS[3][12] := 'W';
DIRS[3][13] := 'WNW';
DIRS[3][14] := 'NW';
DIRS[3][15] := 'NNW';
(*@KEY@: END_WORKSHEET *)
END_FUNCTION_BLOCK

(* ---- SETUP_HOLIDAY_AT.ST ---- *)
(*@PROPERTIES_EX@
TYPE: POU
LOCALE: 0
IEC_LANGUAGE: ST
PLC_TYPE: independent
PROC_TYPE: independent
GROUP: SETUP
*)
(*@KEY@:DESCRIPTION*)

(*@KEY@:END_DESCRIPTION*)
FUNCTION_BLOCK SETUP_HOLIDAY_AT

(*Group:Default*)

VAR_IN_OUT
	HD :	oscat_HOLIDAY_DATA_0_29;
END_VAR

VAR
	init :	BOOL;
END_VAR

(*@KEY@: WORKSHEET
NAME: SETUP_HOLIDAY_AT
IEC_LANGUAGE: ST
*)
(* Daten initialisieren *)
IF init THEN RETURN; END_IF;

init := TRUE;

(* ---- autria --- *)

HD[00].NAME := STRING#'Neujahr';
HD[00].DAY  := SINT#01;
HD[00].MONTH := SINT#01;
HD[00].USE := SINT#01;

HD[01].NAME := STRING#'Heilige Drei Koenige';
HD[01].DAY  := SINT#06;
HD[01].MONTH := SINT#01;
HD[01].USE := SINT#01;

HD[02].NAME := STRING#'Karfreitag';
HD[02].DAY  := SINT#-2;
HD[02].MONTH := SINT#00;
HD[02].USE := SINT#01;

HD[03].NAME := STRING#'Ostersonntag';
HD[03].DAY  := SINT#00;
HD[03].MONTH := SINT#00;
HD[03].USE := SINT#01;

HD[04].NAME := STRING#'Ostermontag';
HD[04].DAY  := SINT#01;
HD[04].MONTH := SINT#00;
HD[04].USE := SINT#01;

HD[05].NAME := STRING#'';
HD[05].DAY  := SINT#01;
HD[05].MONTH := SINT#05;
HD[05].USE := SINT#00;

HD[06].NAME := STRING#'Christi Himmelfahrt';
HD[06].DAY  := SINT#39;
HD[06].MONTH := SINT#00;
HD[06].USE := SINT#01;

HD[07].NAME := STRING#'Pfingstsonntag';
HD[07].DAY  := SINT#49;
HD[07].MONTH := SINT#00;
HD[07].USE := SINT#01;

HD[08].NAME := STRING#'Pfingstmontag';
HD[08].DAY  := SINT#50;
HD[08].MONTH := SINT#00;
HD[08].USE := SINT#01;

HD[09].NAME := STRING#'Fronleichnam';
HD[09].DAY  := SINT#60;
HD[09].MONTH := SINT#00;
HD[09].USE := SINT#01;

HD[10].NAME := STRING#'';
HD[10].DAY  := SINT#08;
HD[10].MONTH := SINT#08;
HD[10].USE := SINT#00;

HD[11].NAME := STRING#'Maria Himmelfahrt';
HD[11].DAY  := SINT#15;
HD[11].MONTH := SINT#08;
HD[11].USE := SINT#01;

HD[12].NAME := STRING#'';
HD[12].DAY  := SINT#03;
HD[12].MONTH := SINT#10;
HD[12].USE := SINT#00;

HD[13].NAME := STRING#'';
HD[13].DAY  := SINT#31;
HD[13].MONTH := SINT#10;
HD[13].USE := SINT#00;

HD[14].NAME := STRING#'Allerheiligen';
HD[14].DAY  := SINT#01;
HD[14].MONTH := SINT#11;
HD[14].USE := SINT#01;

HD[15].NAME := STRING#'Maria Empfängnis';
HD[15].DAY  := SINT#8;
HD[15].MONTH := SINT#12;
HD[15].USE := SINT#01;

HD[16].NAME := STRING#'1. Weihnachtsfeiertag';
HD[16].DAY  := SINT#25;
HD[16].MONTH := SINT#12;
HD[16].USE := SINT#01;

HD[17].NAME := STRING#'2. Weihnachtsfeiertag';
HD[17].DAY  := SINT#26;
HD[17].MONTH := SINT#12;
HD[17].USE := SINT#01;

(*@KEY@: END_WORKSHEET *)
END_FUNCTION_BLOCK

(* ---- SETUP_HOLIDAY_DE.ST ---- *)
(*@PROPERTIES_EX@
TYPE: POU
LOCALE: 0
IEC_LANGUAGE: ST
PLC_TYPE: independent
PROC_TYPE: independent
GROUP: SETUP
*)
(*@KEY@:DESCRIPTION*)

(*@KEY@:END_DESCRIPTION*)
FUNCTION_BLOCK SETUP_HOLIDAY_DE

(*Group:Default*)

VAR_IN_OUT
	HD :	oscat_HOLIDAY_DATA_0_29;
END_VAR

VAR
	init :	BOOL;
END_VAR

(*@KEY@: WORKSHEET
NAME: SETUP_HOLIDAY_DE
IEC_LANGUAGE: ST
*)
(* Daten initialisieren *)
IF init THEN RETURN; END_IF;

init := TRUE;

(* ---- german --- *)

HD[00].NAME := STRING#'Neujahr';
HD[00].DAY  := SINT#01;
HD[00].MONTH := SINT#01;
HD[00].USE := SINT#01;

HD[01].NAME := STRING#'Heilige Drei Koenige';
HD[01].DAY  := SINT#06;
HD[01].MONTH := SINT#01;
HD[01].USE := SINT#01;

HD[02].NAME := STRING#'Karfreitag';
HD[02].DAY  := SINT#-2;
HD[02].MONTH := SINT#00;
HD[02].USE := SINT#01;

HD[03].NAME := STRING#'Ostersonntag';
HD[03].DAY  := SINT#00;
HD[03].MONTH := SINT#00;
HD[03].USE := SINT#01;

HD[04].NAME := STRING#'Ostermontag';
HD[04].DAY  := SINT#01;
HD[04].MONTH := SINT#00;
HD[04].USE := SINT#01;

HD[05].NAME := STRING#'Tag der Arbeit';
HD[05].DAY  := SINT#01;
HD[05].MONTH := SINT#05;
HD[05].USE := SINT#01;

HD[06].NAME := STRING#'Christi Himmelfahrt';
HD[06].DAY  := SINT#39;
HD[06].MONTH := SINT#00;
HD[06].USE := SINT#01;

HD[07].NAME := STRING#'Pfingstsonntag';
HD[07].DAY  := SINT#49;
HD[07].MONTH := SINT#00;
HD[07].USE := SINT#01;

HD[08].NAME := STRING#'Pfingstmontag';
HD[08].DAY  := SINT#50;
HD[08].MONTH := SINT#00;
HD[08].USE := SINT#01;

HD[09].NAME := STRING#'Fronleichnam';
HD[09].DAY  := SINT#60;
HD[09].MONTH := SINT#00;
HD[09].USE := SINT#01;

HD[10].NAME := STRING#'Augsburger Friedensfest';
HD[10].DAY  := SINT#08;
HD[10].MONTH := SINT#08;
HD[10].USE := SINT#00;

HD[11].NAME := STRING#'Maria Himmelfahrt';
HD[11].DAY  := SINT#15;
HD[11].MONTH := SINT#08;
HD[11].USE := SINT#01;

HD[12].NAME := STRING#'Tag der Deutschen Einheit';
HD[12].DAY  := SINT#03;
HD[12].MONTH := SINT#10;
HD[12].USE := SINT#01;

HD[13].NAME := STRING#'Reformationstag';
HD[13].DAY  := SINT#31;
HD[13].MONTH := SINT#10;
HD[13].USE := SINT#00;

HD[14].NAME := STRING#'Allerheiligen';
HD[14].DAY  := SINT#01;
HD[14].MONTH := SINT#11;
HD[14].USE := SINT#01;

HD[15].NAME := STRING#'Buss und Bettag';
HD[15].DAY  := SINT#23;
HD[15].MONTH := SINT#11;
HD[15].USE := SINT#00;

HD[16].NAME := STRING#'1. Weihnachtsfeiertag';
HD[16].DAY  := SINT#25;
HD[16].MONTH := SINT#12;
HD[16].USE := SINT#01;

HD[17].NAME := STRING#'2. Weihnachtsfeiertag';
HD[17].DAY  := SINT#26;
HD[17].MONTH := SINT#12;
HD[17].USE := SINT#01;

(*@KEY@: END_WORKSHEET *)
END_FUNCTION_BLOCK

(* ---- SETUP_HOLIDAY_FR.ST ---- *)
(*@PROPERTIES_EX@
TYPE: POU
LOCALE: 0
IEC_LANGUAGE: ST
PLC_TYPE: independent
PROC_TYPE: independent
GROUP: SETUP
*)
(*@KEY@:DESCRIPTION*)

(*@KEY@:END_DESCRIPTION*)
FUNCTION_BLOCK SETUP_HOLIDAY_FR

(*Group:Default*)

VAR_IN_OUT
	HD :	oscat_HOLIDAY_DATA_0_29;
END_VAR

VAR
	init :	BOOL;
END_VAR

(*@KEY@: WORKSHEET
NAME: SETUP_HOLIDAY_FR
IEC_LANGUAGE: ST
*)
(* Daten initialisieren *)
IF init THEN RETURN; END_IF;

init := TRUE;

(* ---- france --- *)

HD[00].NAME := STRING#'Nouvel an';
HD[00].DAY  := SINT#01;
HD[00].MONTH := SINT#01;
HD[00].USE := SINT#01;

HD[01].NAME := STRING#'St Valentin';
HD[01].DAY  := SINT#14;
HD[01].MONTH := SINT#02;
HD[01].USE := SINT#00;

HD[02].NAME := STRING#'Vendredi Saint (alsace)';
HD[02].DAY  := SINT#-2;
HD[02].MONTH := SINT#00;
HD[02].USE := SINT#00;

HD[03].NAME := STRING#'Dimanche de pâques';
HD[03].DAY  := SINT#00;
HD[03].MONTH := SINT#00;
HD[03].USE := SINT#01;

HD[04].NAME := STRING#'Lundi de pâques';
HD[04].DAY  := SINT#01;
HD[04].MONTH := SINT#00;
HD[04].USE := SINT#01;

HD[05].NAME := STRING#'Jeudi de Ascension';
HD[05].DAY  := SINT#39;
HD[05].MONTH := SINT#00;
HD[05].USE := SINT#01;

HD[06].NAME := STRING#'dimanche de Pentecôte';
HD[06].DAY  := SINT#49;
HD[06].MONTH := SINT#00;
HD[06].USE := SINT#01;

HD[07].NAME := STRING#'jeudi de la Trinité';
HD[07].DAY  := SINT#60;
HD[07].MONTH := SINT#00;
HD[07].USE := SINT#00;

HD[08].NAME := STRING#'Fête du travail';
HD[08].DAY  := SINT#01;
HD[08].MONTH := SINT#05;
HD[08].USE := SINT#01;

HD[09].NAME := STRING#'Victoire 1945 ';
HD[09].DAY  := SINT#08;
HD[09].MONTH := SINT#05;
HD[09].USE := SINT#01;

HD[10].NAME := STRING#'Prise de La bastille';
HD[10].DAY  := SINT#14;
HD[10].MONTH := SINT#07;
HD[10].USE := SINT#01;

HD[11].NAME := STRING#'15 Août 1944';
HD[11].DAY  := SINT#15;
HD[11].MONTH := SINT#08;
HD[11].USE := SINT#01;

HD[12].NAME := STRING#'Halloween';
HD[12].DAY  := SINT#31;
HD[12].MONTH := SINT#10;
HD[12].USE := SINT#00;

HD[13].NAME := STRING#'Armistice 1918';
HD[13].DAY  := SINT#11;
HD[13].MONTH := SINT#11;
HD[13].USE := SINT#01;

HD[14].NAME := STRING#'Noël';
HD[14].DAY  := SINT#25;
HD[14].MONTH := SINT#12;
HD[14].USE := SINT#01;

HD[15].NAME := STRING#'Saint Étienne (alsace)';
HD[15].DAY  := SINT#26;
HD[15].MONTH := SINT#12;
HD[15].USE := SINT#00;

HD[16].NAME := STRING#'Fête de la musique';
HD[16].DAY  := SINT#21;
HD[16].MONTH := SINT#06;
HD[16].USE := SINT#00;
(*@KEY@: END_WORKSHEET *)
END_FUNCTION_BLOCK

(* ---- SETUP_LANGUAGE.ST ---- *)
(*@PROPERTIES_EX@
TYPE: POU
LOCALE: 0
IEC_LANGUAGE: ST
PLC_TYPE: independent
PROC_TYPE: independent
GROUP: SETUP
*)
(*@KEY@:DESCRIPTION*)

(*@KEY@:END_DESCRIPTION*)
FUNCTION_BLOCK SETUP_LANGUAGE

(*Group:Default*)

VAR_IN_OUT
	LANGUAGE :	oscat_LANGUAGE;
END_VAR

VAR
	init :	BOOL;
END_VAR

(*@KEY@: WORKSHEET
NAME: SETUP_LANGUAGE
IEC_LANGUAGE: ST
*)
(* Daten initialisieren *)
IF init THEN RETURN; END_IF;
init := TRUE;

LANGUAGE.DEFAULT  := 1; (* 1=english, 2=german 3=french *)
LANGUAGE.LMAX := 3;
(*@KEY@: END_WORKSHEET *)
END_FUNCTION_BLOCK

(* ---- SETUP_LOCATION.ST ---- *)
(*@PROPERTIES_EX@
TYPE: POU
LOCALE: 0
IEC_LANGUAGE: ST
PLC_TYPE: independent
PROC_TYPE: independent
GROUP: SETUP
*)
(*@KEY@:DESCRIPTION*)

(*@KEY@:END_DESCRIPTION*)
FUNCTION_BLOCK SETUP_LOCATION

(*Group:Default*)

VAR_IN_OUT
	LOCATION :	oscat_LOCATION;
END_VAR

VAR
	init :	BOOL;
END_VAR

(*@KEY@: WORKSHEET
NAME: SETUP_LOCATION
IEC_LANGUAGE: ST
*)
(* Daten initialisieren *)
IF init THEN RETURN; END_IF;
init := TRUE;

LOCATION.DEFAULT  := 1;  (* 1=germany, 2=austria 3=france 4=belgium-german 5= italien-Südtirol *)
LOCATION.LMAX := 5;

LOCATION.LANGUAGE[1] := 2;
LOCATION.LANGUAGE[2] := 2;
LOCATION.LANGUAGE[3] := 3;
LOCATION.LANGUAGE[4] := 2;
LOCATION.LANGUAGE[5] := 2;

(*@KEY@: END_WORKSHEET *)
END_FUNCTION_BLOCK

(* ---- SETUP_MONTHS.ST ---- *)
(*@PROPERTIES_EX@
TYPE: POU
LOCALE: 0
IEC_LANGUAGE: ST
PLC_TYPE: independent
PROC_TYPE: independent
GROUP: SETUP
*)
(*@KEY@:DESCRIPTION*)

(*@KEY@:END_DESCRIPTION*)
FUNCTION_BLOCK SETUP_MONTHS

(*Group:Default*)

VAR_IN_OUT
	MONTHS :	oscat_MONTHS;
END_VAR

VAR
	init :	BOOL;
END_VAR

(*@KEY@: WORKSHEET
NAME: SETUP_MONTHS
IEC_LANGUAGE: ST
*)
(* Daten initialisieren *)
IF init THEN RETURN; END_IF;
init := TRUE;

(* ---- english --- *)
MONTHS[1][01] := 'January';
MONTHS[1][02] := 'February';
MONTHS[1][03] := 'March';
MONTHS[1][04] := 'April';
MONTHS[1][05] := 'May';
MONTHS[1][06] := 'June';
MONTHS[1][07] := 'July';
MONTHS[1][08] := 'August';
MONTHS[1][09] := 'September';
MONTHS[1][10] := 'October';
MONTHS[1][11] := 'November';
MONTHS[1][12] := 'December';

(* ---- german --- *)
MONTHS[2][01] := 'Januar';
MONTHS[2][02] := 'Februar';
MONTHS[2][03] := 'März';
MONTHS[2][04] := 'April';
MONTHS[2][05] := 'Mai';
MONTHS[2][06] := 'Juni';
MONTHS[2][07] := 'Juli';
MONTHS[2][08] := 'August';
MONTHS[2][09] := 'September';
MONTHS[2][10] := 'Oktober';
MONTHS[2][11] := 'November';
MONTHS[2][12] := 'Dezember';

(* ---- french --- *)
MONTHS[3][01] := 'Janvier';
MONTHS[3][02] := 'Février';
MONTHS[3][03] := 'mars';
MONTHS[3][04] := 'Avril';
MONTHS[3][05] := 'Mai';
MONTHS[3][06] := 'Juin';
MONTHS[3][07] := 'Juillet';
MONTHS[3][08] := 'Août';
MONTHS[3][09] := 'Septembre';
MONTHS[3][10] := 'Octobre';
MONTHS[3][11] := 'Novembre';
MONTHS[3][12] := 'Decembre';
(*@KEY@: END_WORKSHEET *)
END_FUNCTION_BLOCK
